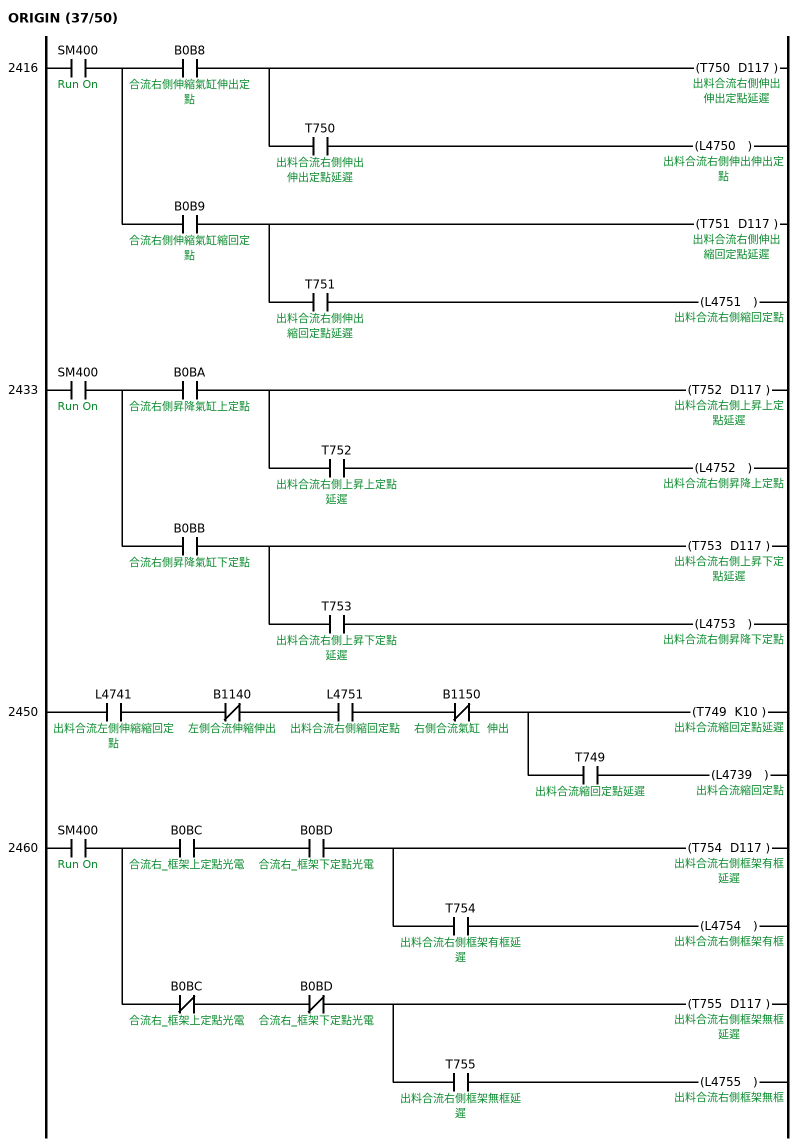
[picture p456: ladder of ORIGIN, rungs at steps 2416 to 2460]
2416  LD      SM400  ; Run On
      MPS
      AND     B0B8  ; 合流右側伸縮氣缸伸出定點
      OUT     T750 D117  ; 出料合流右側伸出 伸出定點延遲
      AND     T750  ; 出料合流右側伸出 伸出定點延遲
      OUT     L4750  ; 出料合流右側伸出伸出定點
      MPP
      AND     B0B9  ; 合流右側伸縮氣缸縮回定點
      OUT     T751 D117  ; 出料合流右側伸出 縮回定點延遲
      AND     T751  ; 出料合流右側伸出 縮回定點延遲
      OUT     L4751  ; 出料合流右側縮回定點
2433  LD      SM400  ; Run On
      MPS
      AND     B0BA  ; 合流右側昇降氣缸上定點
      OUT     T752 D117  ; 出料合流右側上昇上定點延遲
      AND     T752  ; 出料合流右側上昇上定點延遲
      OUT     L4752  ; 出料合流右側昇降上定點
      MPP
      AND     B0BB  ; 合流右側昇降氣缸下定點
      OUT     T753 D117  ; 出料合流右側上昇下定點延遲
      AND     T753  ; 出料合流右側上昇下定點延遲
      OUT     L4753  ; 出料合流右側昇降下定點
2450  LD      L4741  ; 出料合流左側伸縮縮回定點
      ANI     B1140  ; 左側合流伸縮伸出
      AND     L4751  ; 出料合流右側縮回定點
      ANI     B1150  ; 右側合流氣缸  伸出
      OUT     T749 K10  ; 出料合流縮回定點延遲
      AND     T749  ; 出料合流縮回定點延遲
      OUT     L4739  ; 出料合流縮回定點
2460  LD      SM400  ; Run On
      MPS
      AND     B0BC  ; 合流右_框架上定點光電
      AND     B0BD  ; 合流右_框架下定點光電
      OUT     T754 D117  ; 出料合流右側框架有框延遲
      AND     T754  ; 出料合流右側框架有框延遲
      OUT     L4754  ; 出料合流右側框架有框
      MPP
      ANI     B0BC  ; 合流右_框架上定點光電
      ANI     B0BD  ; 合流右_框架下定點光電
      OUT     T755 D117  ; 出料合流右側框架無框延遲
      AND     T755  ; 出料合流右側框架無框延遲
      OUT     L4755  ; 出料合流右側框架無框
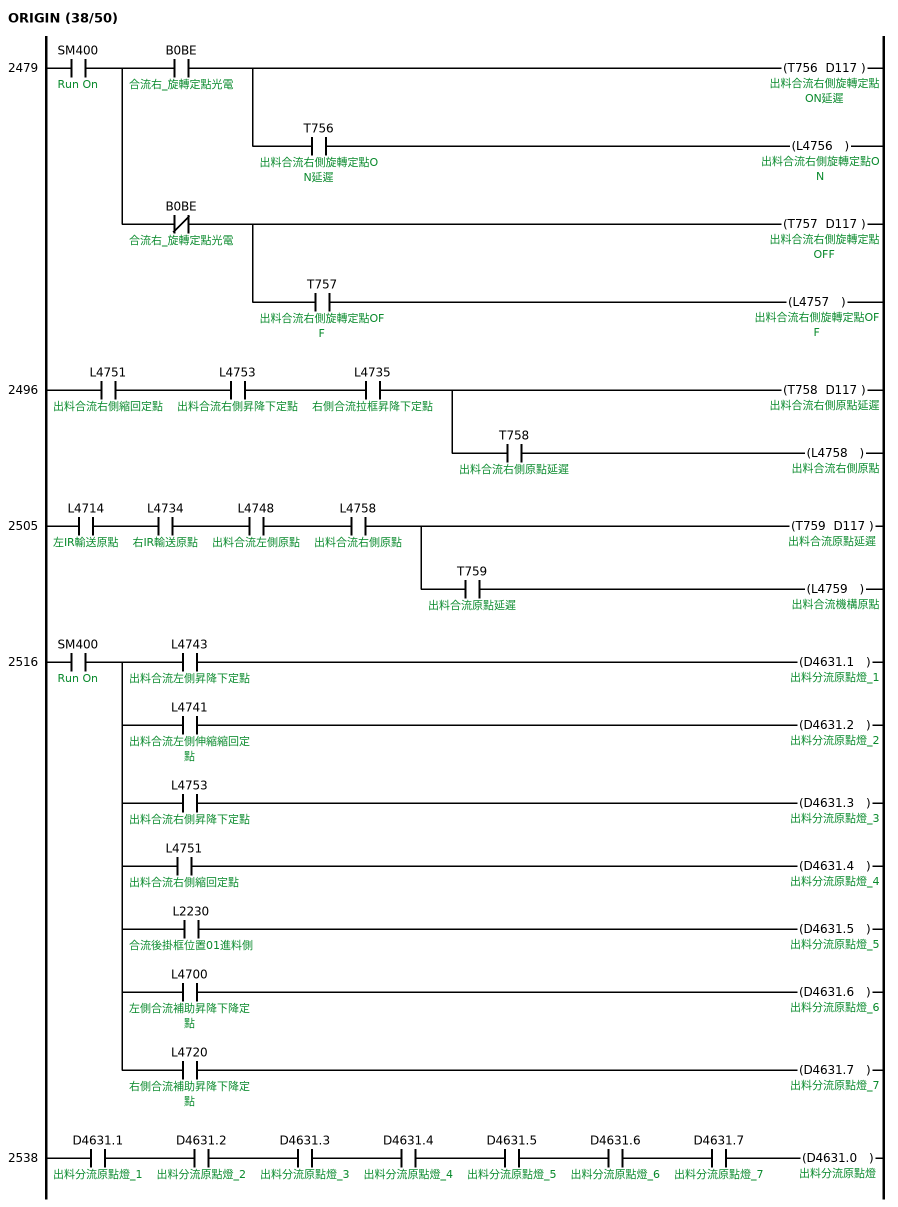
2479  LD      SM400  ; Run On
      MPS
      AND     B0BE  ; 合流右_旋轉定點光電
      OUT     T756 D117  ; 出料合流右側旋轉定點ON延遲
      AND     T756  ; 出料合流右側旋轉定點ON延遲
      OUT     L4756  ; 出料合流右側旋轉定點ON
      MPP
      ANI     B0BE  ; 合流右_旋轉定點光電
      OUT     T757 D117  ; 出料合流右側旋轉定點OFF
      AND     T757  ; 出料合流右側旋轉定點OFF
      OUT     L4757  ; 出料合流右側旋轉定點OFF
2496  LD      L4751  ; 出料合流右側縮回定點
      AND     L4753  ; 出料合流右側昇降下定點
      AND     L4735  ; 右側合流拉框昇降下定點
      OUT     T758 D117  ; 出料合流右側原點延遲
      AND     T758  ; 出料合流右側原點延遲
      OUT     L4758  ; 出料合流右側原點
2505  LD      L4714  ; 左IR輸送原點
      AND     L4734  ; 右IR輸送原點
      AND     L4748  ; 出料合流左側原點
      AND     L4758  ; 出料合流右側原點
      OUT     T759 D117  ; 出料合流原點延遲
      AND     T759  ; 出料合流原點延遲
      OUT     L4759  ; 出料合流機構原點
2516  LD      SM400  ; Run On
      MPS
      AND     L4743  ; 出料合流左側昇降下定點
      OUT     D4631.1  ; 出料分流原點燈_1
      MRD
      AND     L4741  ; 出料合流左側伸縮縮回定點
      OUT     D4631.2  ; 出料分流原點燈_2
      MRD
      AND     L4753  ; 出料合流右側昇降下定點
      OUT     D4631.3  ; 出料分流原點燈_3
      MRD
      AND     L4751  ; 出料合流右側縮回定點
      OUT     D4631.4  ; 出料分流原點燈_4
      MRD
      AND     L2230  ; 合流後掛框位置01進料側
      OUT     D4631.5  ; 出料分流原點燈_5
      MRD
      AND     L4700  ; 左側合流補助昇降下降定點
      OUT     D4631.6  ; 出料分流原點燈_6
      MPP
      AND     L4720  ; 右側合流補助昇降下降定點
      OUT     D4631.7  ; 出料分流原點燈_7
2538  LD      D4631.1  ; 出料分流原點燈_1
      AND     D4631.2  ; 出料分流原點燈_2
      AND     D4631.3  ; 出料分流原點燈_3
      AND     D4631.4  ; 出料分流原點燈_4
      AND     D4631.5  ; 出料分流原點燈_5
      AND     D4631.6  ; 出料分流原點燈_6
      AND     D4631.7  ; 出料分流原點燈_7
      OUT     D4631.0  ; 出料分流原點燈
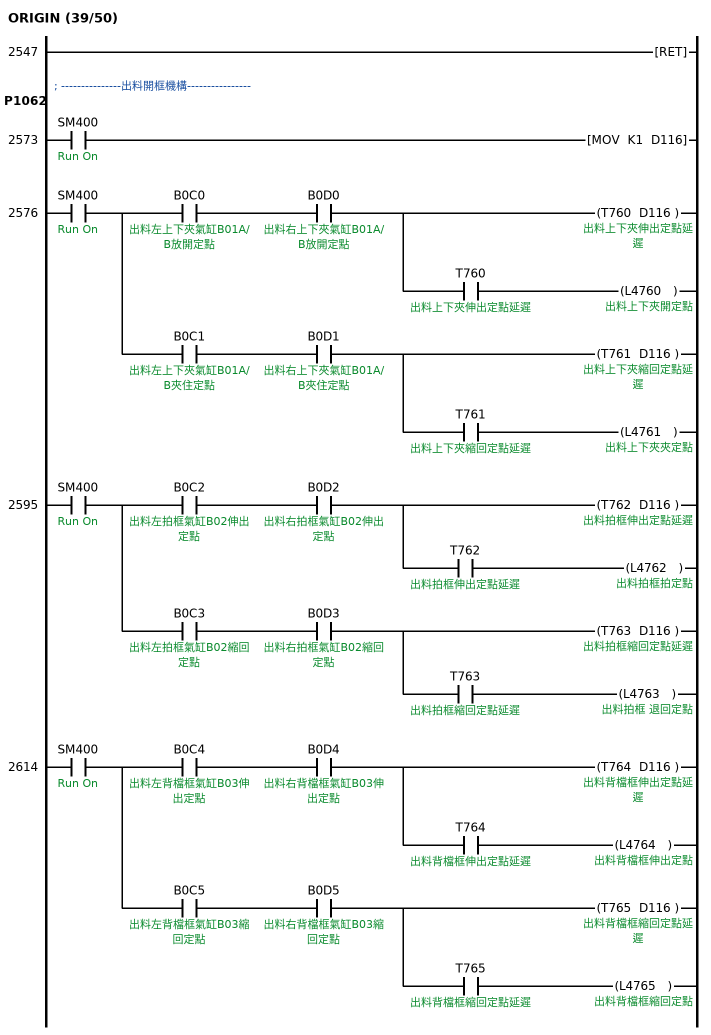
2547  RET
; ---------------出料開框機構----------------
      P1062
2573  LD      SM400  ; Run On
      MOV     K1 D116
2576  LD      SM400  ; Run On
      MPS
      AND     B0C0  ; 出料左上下夾氣缸B01A/B放開定點
      AND     B0D0  ; 出料右上下夾氣缸B01A/B放開定點
      OUT     T760 D116  ; 出料上下夾伸出定點延遲
      AND     T760  ; 出料上下夾伸出定點延遲
      OUT     L4760  ; 出料上下夾開定點
      MPP
      AND     B0C1  ; 出料左上下夾氣缸B01A/B夾住定點
      AND     B0D1  ; 出料右上下夾氣缸B01A/B夾住定點
      OUT     T761 D116  ; 出料上下夾縮回定點延遲
      AND     T761  ; 出料上下夾縮回定點延遲
      OUT     L4761  ; 出料上下夾夾定點
2595  LD      SM400  ; Run On
      MPS
      AND     B0C2  ; 出料左拍框氣缸B02伸出定點
      AND     B0D2  ; 出料右拍框氣缸B02伸出定點
      OUT     T762 D116  ; 出料拍框伸出定點延遲
      AND     T762  ; 出料拍框伸出定點延遲
      OUT     L4762  ; 出料拍框拍定點
      MPP
      AND     B0C3  ; 出料左拍框氣缸B02縮回定點
      AND     B0D3  ; 出料右拍框氣缸B02縮回定點
      OUT     T763 D116  ; 出料拍框縮回定點延遲
      AND     T763  ; 出料拍框縮回定點延遲
      OUT     L4763  ; 出料拍框 退回定點
2614  LD      SM400  ; Run On
      MPS
      AND     B0C4  ; 出料左背檔框氣缸B03伸出定點
      AND     B0D4  ; 出料右背檔框氣缸B03伸出定點
      OUT     T764 D116  ; 出料背檔框伸出定點延遲
      AND     T764  ; 出料背檔框伸出定點延遲
      OUT     L4764  ; 出料背檔框伸出定點
      MPP
      AND     B0C5  ; 出料左背檔框氣缸B03縮回定點
      AND     B0D5  ; 出料右背檔框氣缸B03縮回定點
      OUT     T765 D116  ; 出料背檔框縮回定點延遲
      AND     T765  ; 出料背檔框縮回定點延遲
      OUT     L4765  ; 出料背檔框縮回定點
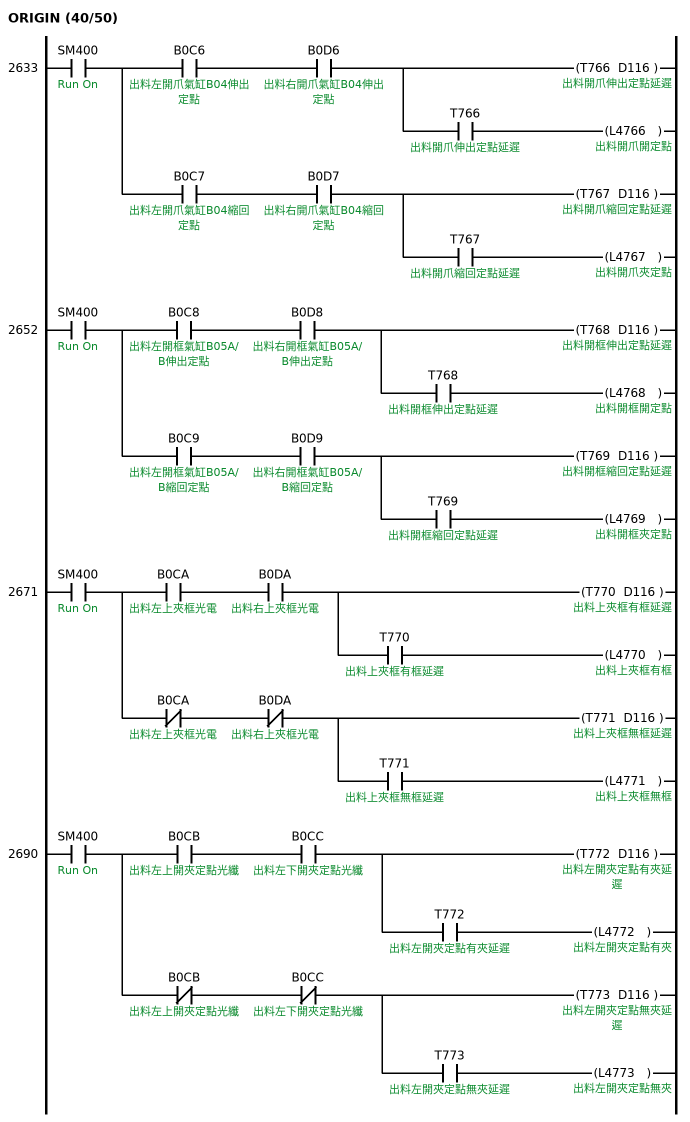
2633  LD      SM400  ; Run On
      MPS
      AND     B0C6  ; 出料左開爪氣缸B04伸出定點
      AND     B0D6  ; 出料右開爪氣缸B04伸出定點
      OUT     T766 D116  ; 出料開爪伸出定點延遲
      AND     T766  ; 出料開爪伸出定點延遲
      OUT     L4766  ; 出料開爪開定點
      MPP
      AND     B0C7  ; 出料左開爪氣缸B04縮回定點
      AND     B0D7  ; 出料右開爪氣缸B04縮回定點
      OUT     T767 D116  ; 出料開爪縮回定點延遲
      AND     T767  ; 出料開爪縮回定點延遲
      OUT     L4767  ; 出料開爪夾定點
2652  LD      SM400  ; Run On
      MPS
      AND     B0C8  ; 出料左開框氣缸B05A/B伸出定點
      AND     B0D8  ; 出料右開框氣缸B05A/B伸出定點
      OUT     T768 D116  ; 出料開框伸出定點延遲
      AND     T768  ; 出料開框伸出定點延遲
      OUT     L4768  ; 出料開框開定點
      MPP
      AND     B0C9  ; 出料左開框氣缸B05A/B縮回定點
      AND     B0D9  ; 出料右開框氣缸B05A/B縮回定點
      OUT     T769 D116  ; 出料開框縮回定點延遲
      AND     T769  ; 出料開框縮回定點延遲
      OUT     L4769  ; 出料開框夾定點
2671  LD      SM400  ; Run On
      MPS
      AND     B0CA  ; 出料左上夾框光電
      AND     B0DA  ; 出料右上夾框光電
      OUT     T770 D116  ; 出料上夾框有框延遲
      AND     T770  ; 出料上夾框有框延遲
      OUT     L4770  ; 出料上夾框有框
      MPP
      ANI     B0CA  ; 出料左上夾框光電
      ANI     B0DA  ; 出料右上夾框光電
      OUT     T771 D116  ; 出料上夾框無框延遲
      AND     T771  ; 出料上夾框無框延遲
      OUT     L4771  ; 出料上夾框無框
2690  LD      SM400  ; Run On
      MPS
      AND     B0CB  ; 出料左上開夾定點光纖
      AND     B0CC  ; 出料左下開夾定點光纖
      OUT     T772 D116  ; 出料左開夾定點有夾延遲
      AND     T772  ; 出料左開夾定點有夾延遲
      OUT     L4772  ; 出料左開夾定點有夾
      MPP
      ANI     B0CB  ; 出料左上開夾定點光纖
      ANI     B0CC  ; 出料左下開夾定點光纖
      OUT     T773 D116  ; 出料左開夾定點無夾延遲
      AND     T773  ; 出料左開夾定點無夾延遲
      OUT     L4773  ; 出料左開夾定點無夾
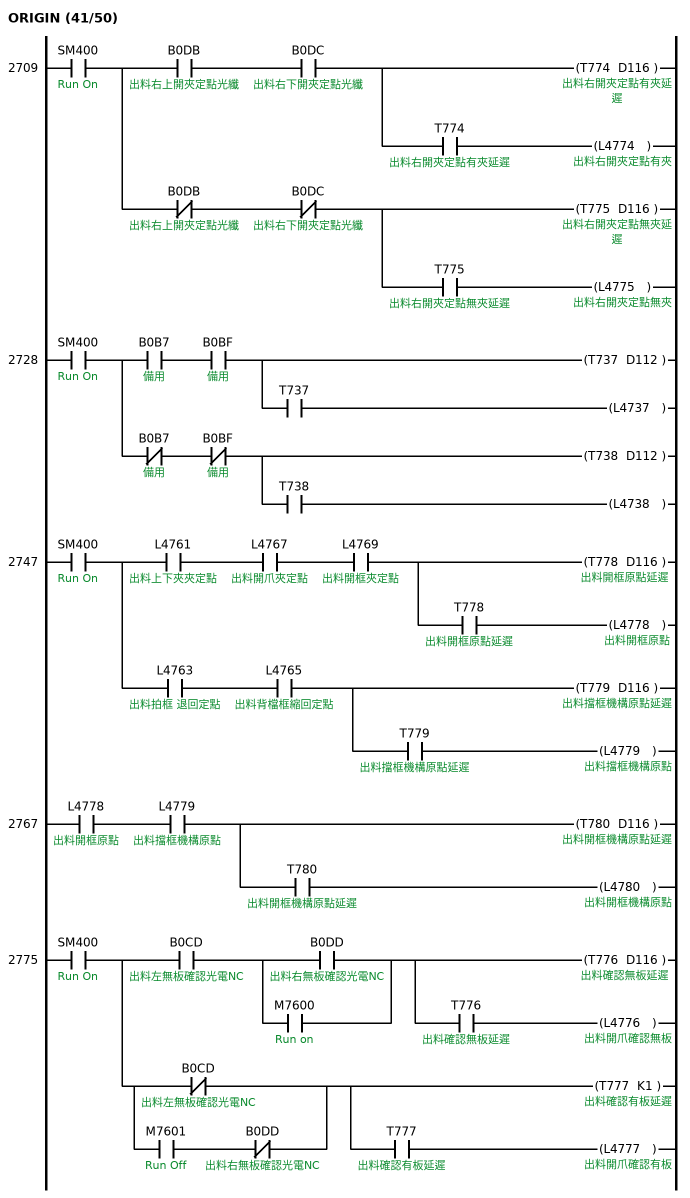
2709  LD      SM400  ; Run On
      MPS
      AND     B0DB  ; 出料右上開夾定點光纖
      AND     B0DC  ; 出料右下開夾定點光纖
      OUT     T774 D116  ; 出料右開夾定點有夾延遲
      AND     T774  ; 出料右開夾定點有夾延遲
      OUT     L4774  ; 出料右開夾定點有夾
      MPP
      ANI     B0DB  ; 出料右上開夾定點光纖
      ANI     B0DC  ; 出料右下開夾定點光纖
      OUT     T775 D116  ; 出料右開夾定點無夾延遲
      AND     T775  ; 出料右開夾定點無夾延遲
      OUT     L4775  ; 出料右開夾定點無夾
2728  LD      SM400  ; Run On
      MPS
      AND     B0B7  ; 備用
      AND     B0BF  ; 備用
      OUT     T737 D112
      AND     T737
      OUT     L4737
      MPP
      ANI     B0B7  ; 備用
      ANI     B0BF  ; 備用
      OUT     T738 D112
      AND     T738
      OUT     L4738
2747  LD      SM400  ; Run On
      MPS
      AND     L4761  ; 出料上下夾夾定點
      AND     L4767  ; 出料開爪夾定點
      AND     L4769  ; 出料開框夾定點
      OUT     T778 D116  ; 出料開框原點延遲
      AND     T778  ; 出料開框原點延遲
      OUT     L4778  ; 出料開框原點
      MPP
      AND     L4763  ; 出料拍框 退回定點
      AND     L4765  ; 出料背檔框縮回定點
      OUT     T779 D116  ; 出料擋框機構原點延遲
      AND     T779  ; 出料擋框機構原點延遲
      OUT     L4779  ; 出料擋框機構原點
2767  LD      L4778  ; 出料開框原點
      AND     L4779  ; 出料擋框機構原點
      OUT     T780 D116  ; 出料開框機構原點延遲
      AND     T780  ; 出料開框機構原點延遲
      OUT     L4780  ; 出料開框機構原點
2775  LD      SM400  ; Run On
      MPS
      AND     B0CD  ; 出料左無板確認光電NC
      LD      B0DD  ; 出料右無板確認光電NC
      OR      M7600  ; Run on
      ANB
      OUT     T776 D116  ; 出料確認無板延遲
      AND     T776  ; 出料確認無板延遲
      OUT     L4776  ; 出料開爪確認無板
      MPP
      LDI     B0CD  ; 出料左無板確認光電NC
      LD      M7601  ; Run Off
      ANI     B0DD  ; 出料右無板確認光電NC
      ORB
      ANB
      OUT     T777 K1  ; 出料確認有板延遲
      AND     T777  ; 出料確認有板延遲
      OUT     L4777  ; 出料開爪確認有板
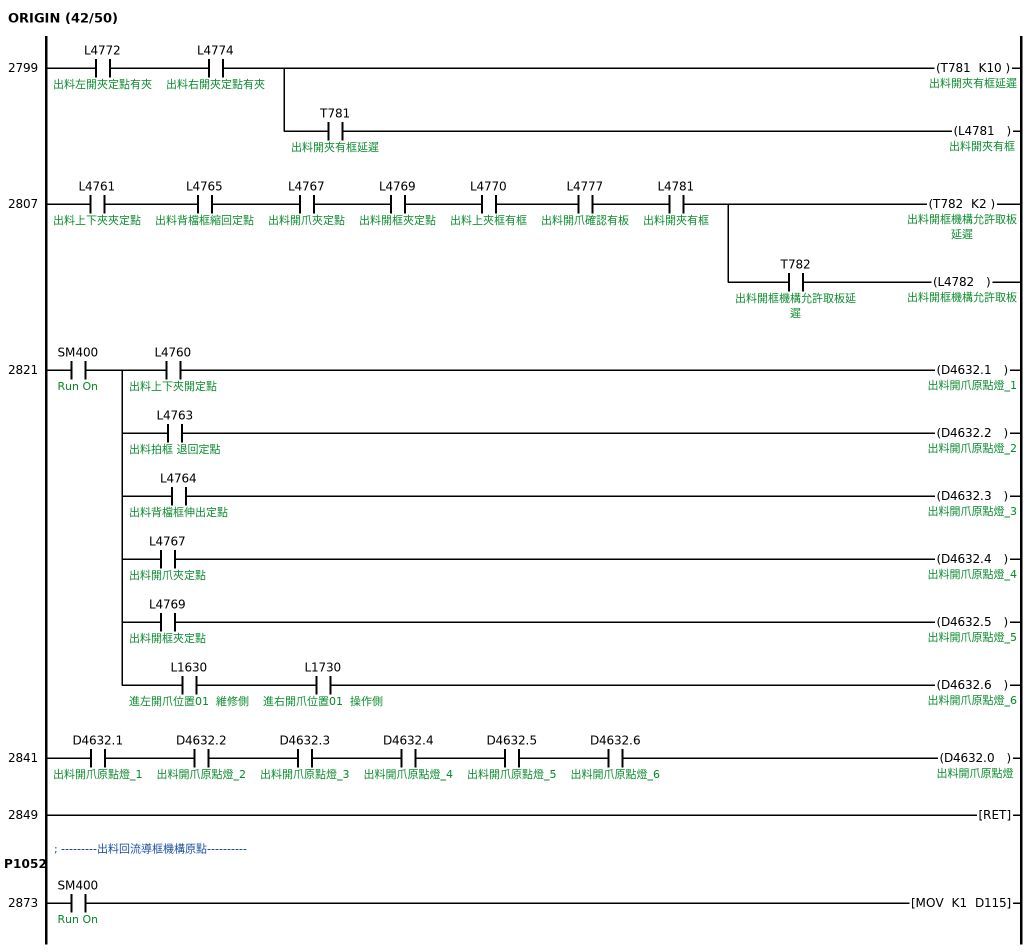
2799  LD      L4772  ; 出料左開夾定點有夾
      AND     L4774  ; 出料右開夾定點有夾
      OUT     T781 K10  ; 出料開夾有框延遲
      AND     T781  ; 出料開夾有框延遲
      OUT     L4781  ; 出料開夾有框
2807  LD      L4761  ; 出料上下夾夾定點
      AND     L4765  ; 出料背檔框縮回定點
      AND     L4767  ; 出料開爪夾定點
      AND     L4769  ; 出料開框夾定點
      AND     L4770  ; 出料上夾框有框
      AND     L4777  ; 出料開爪確認有板
      AND     L4781  ; 出料開夾有框
      OUT     T782 K2  ; 出料開框機構允許取板延遲
      AND     T782  ; 出料開框機構允許取板延遲
      OUT     L4782  ; 出料開框機構允許取板
2821  LD      SM400  ; Run On
      MPS
      AND     L4760  ; 出料上下夾開定點
      OUT     D4632.1  ; 出料開爪原點燈_1
      MRD
      AND     L4763  ; 出料拍框 退回定點
      OUT     D4632.2  ; 出料開爪原點燈_2
      MRD
      AND     L4764  ; 出料背檔框伸出定點
      OUT     D4632.3  ; 出料開爪原點燈_3
      MRD
      AND     L4767  ; 出料開爪夾定點
      OUT     D4632.4  ; 出料開爪原點燈_4
      MRD
      AND     L4769  ; 出料開框夾定點
      OUT     D4632.5  ; 出料開爪原點燈_5
      MPP
      AND     L1630  ; 進左開爪位置01  維修側
      AND     L1730  ; 進右開爪位置01  操作側
      OUT     D4632.6  ; 出料開爪原點燈_6
2841  LD      D4632.1  ; 出料開爪原點燈_1
      AND     D4632.2  ; 出料開爪原點燈_2
      AND     D4632.3  ; 出料開爪原點燈_3
      AND     D4632.4  ; 出料開爪原點燈_4
      AND     D4632.5  ; 出料開爪原點燈_5
      AND     D4632.6  ; 出料開爪原點燈_6
      OUT     D4632.0  ; 出料開爪原點燈
2849  RET
; ---------出料回流導框機構原點----------
      P1052
2873  LD      SM400  ; Run On
      MOV     K1 D115
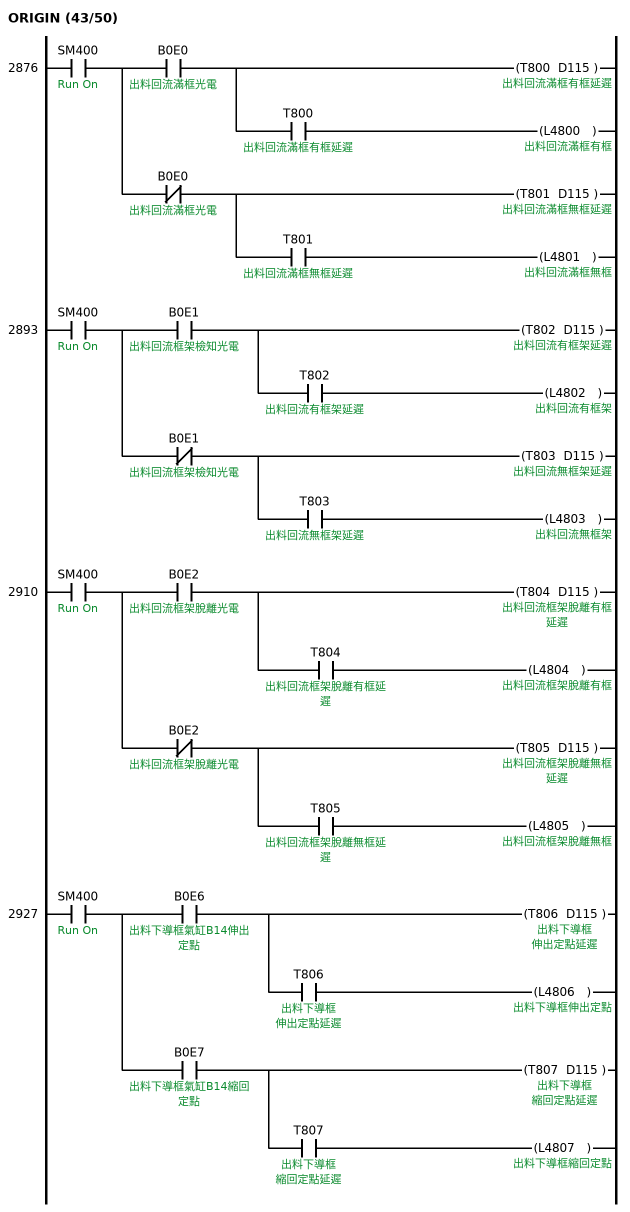
2876  LD      SM400  ; Run On
      MPS
      AND     B0E0  ; 出料回流滿框光電
      OUT     T800 D115  ; 出料回流滿框有框延遲
      AND     T800  ; 出料回流滿框有框延遲
      OUT     L4800  ; 出料回流滿框有框
      MPP
      ANI     B0E0  ; 出料回流滿框光電
      OUT     T801 D115  ; 出料回流滿框無框延遲
      AND     T801  ; 出料回流滿框無框延遲
      OUT     L4801  ; 出料回流滿框無框
2893  LD      SM400  ; Run On
      MPS
      AND     B0E1  ; 出料回流框架檢知光電
      OUT     T802 D115  ; 出料回流有框架延遲
      AND     T802  ; 出料回流有框架延遲
      OUT     L4802  ; 出料回流有框架
      MPP
      ANI     B0E1  ; 出料回流框架檢知光電
      OUT     T803 D115  ; 出料回流無框架延遲
      AND     T803  ; 出料回流無框架延遲
      OUT     L4803  ; 出料回流無框架
2910  LD      SM400  ; Run On
      MPS
      AND     B0E2  ; 出料回流框架脫離光電
      OUT     T804 D115  ; 出料回流框架脫離有框延遲
      AND     T804  ; 出料回流框架脫離有框延遲
      OUT     L4804  ; 出料回流框架脫離有框
      MPP
      ANI     B0E2  ; 出料回流框架脫離光電
      OUT     T805 D115  ; 出料回流框架脫離無框延遲
      AND     T805  ; 出料回流框架脫離無框延遲
      OUT     L4805  ; 出料回流框架脫離無框
2927  LD      SM400  ; Run On
      MPS
      AND     B0E6  ; 出料下導框氣缸B14伸出定點
      OUT     T806 D115  ; 出料下導框    伸出定點延遲
      AND     T806  ; 出料下導框    伸出定點延遲
      OUT     L4806  ; 出料下導框伸出定點
      MPP
      AND     B0E7  ; 出料下導框氣缸B14縮回定點
      OUT     T807 D115  ; 出料下導框    縮回定點延遲
      AND     T807  ; 出料下導框    縮回定點延遲
      OUT     L4807  ; 出料下導框縮回定點
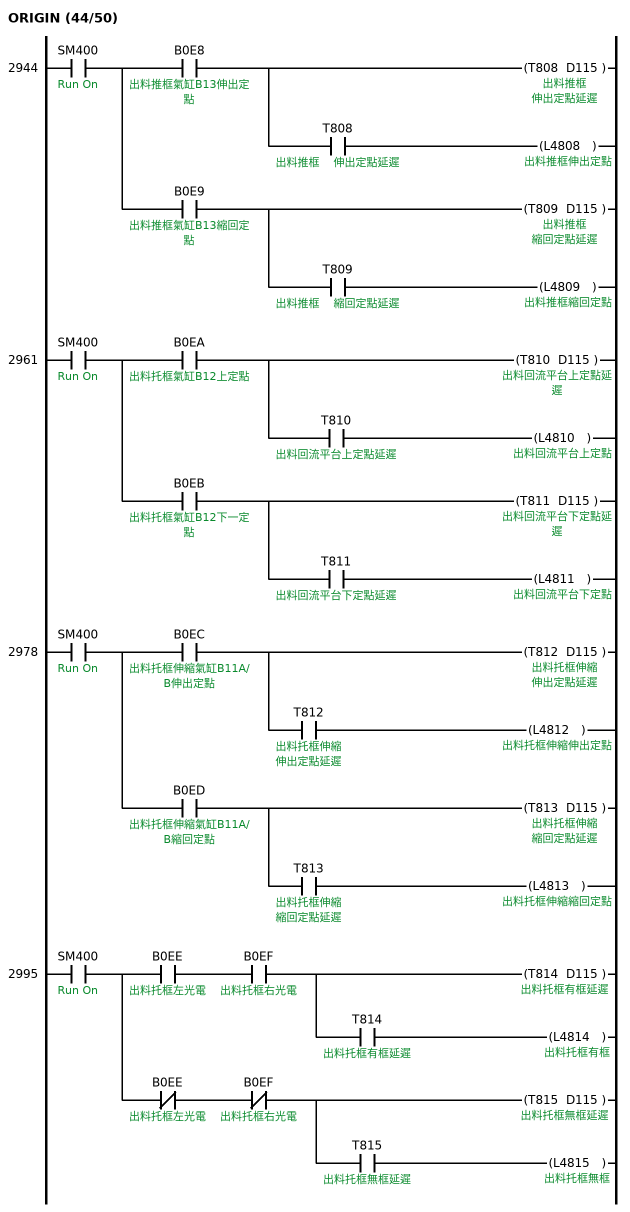
2944  LD      SM400  ; Run On
      MPS
      AND     B0E8  ; 出料推框氣缸B13伸出定點
      OUT     T808 D115  ; 出料推框    伸出定點延遲
      AND     T808  ; 出料推框    伸出定點延遲
      OUT     L4808  ; 出料推框伸出定點
      MPP
      AND     B0E9  ; 出料推框氣缸B13縮回定點
      OUT     T809 D115  ; 出料推框    縮回定點延遲
      AND     T809  ; 出料推框    縮回定點延遲
      OUT     L4809  ; 出料推框縮回定點
2961  LD      SM400  ; Run On
      MPS
      AND     B0EA  ; 出料托框氣缸B12上定點
      OUT     T810 D115  ; 出料回流平台上定點延遲
      AND     T810  ; 出料回流平台上定點延遲
      OUT     L4810  ; 出料回流平台上定點
      MPP
      AND     B0EB  ; 出料托框氣缸B12下一定點
      OUT     T811 D115  ; 出料回流平台下定點延遲
      AND     T811  ; 出料回流平台下定點延遲
      OUT     L4811  ; 出料回流平台下定點
2978  LD      SM400  ; Run On
      MPS
      AND     B0EC  ; 出料托框伸縮氣缸B11A/B伸出定點
      OUT     T812 D115  ; 出料托框伸縮    伸出定點延遲
      AND     T812  ; 出料托框伸縮    伸出定點延遲
      OUT     L4812  ; 出料托框伸縮伸出定點
      MPP
      AND     B0ED  ; 出料托框伸縮氣缸B11A/B縮回定點
      OUT     T813 D115  ; 出料托框伸縮    縮回定點延遲
      AND     T813  ; 出料托框伸縮    縮回定點延遲
      OUT     L4813  ; 出料托框伸縮縮回定點
2995  LD      SM400  ; Run On
      MPS
      AND     B0EE  ; 出料托框左光電
      AND     B0EF  ; 出料托框右光電
      OUT     T814 D115  ; 出料托框有框延遲
      AND     T814  ; 出料托框有框延遲
      OUT     L4814  ; 出料托框有框
      MPP
      ANI     B0EE  ; 出料托框左光電
      ANI     B0EF  ; 出料托框右光電
      OUT     T815 D115  ; 出料托框無框延遲
      AND     T815  ; 出料托框無框延遲
      OUT     L4815  ; 出料托框無框
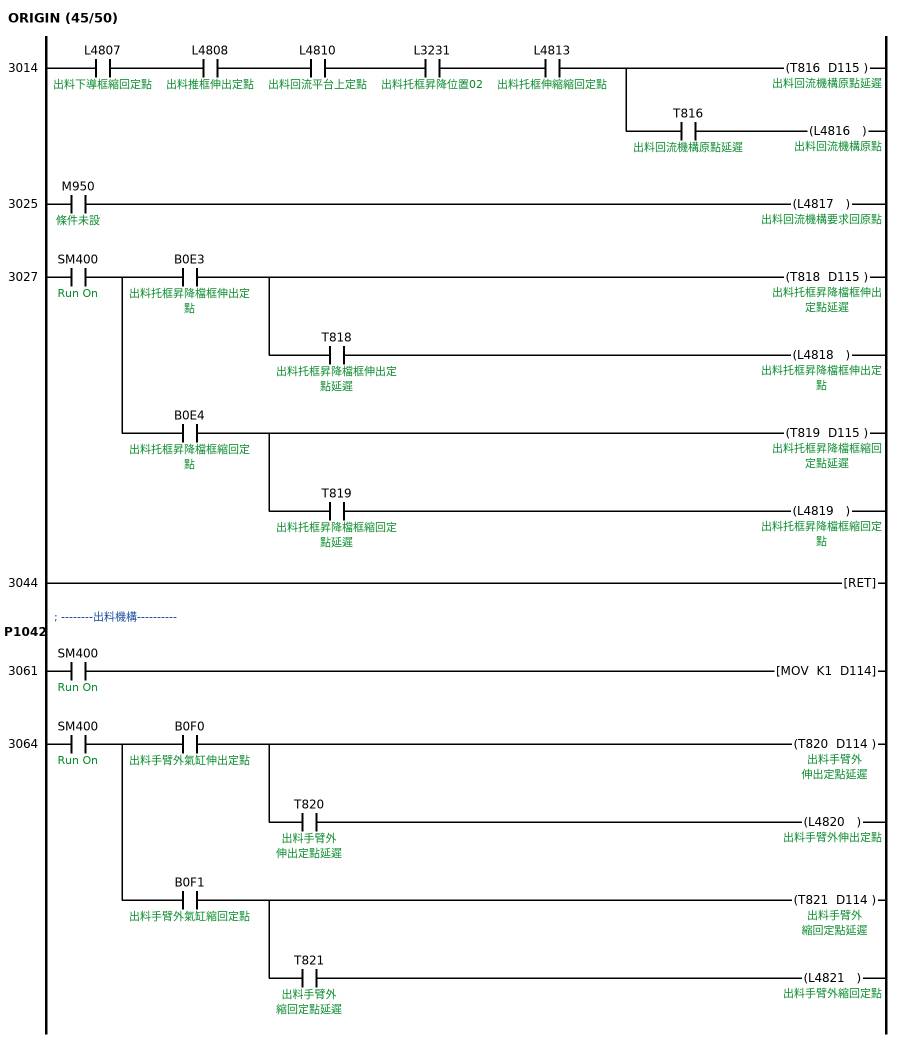
3014  LD      L4807  ; 出料下導框縮回定點
      AND     L4808  ; 出料推框伸出定點
      AND     L4810  ; 出料回流平台上定點
      AND     L3231  ; 出料托框昇降位置02
      AND     L4813  ; 出料托框伸縮縮回定點
      OUT     T816 D115  ; 出料回流機構原點延遲
      AND     T816  ; 出料回流機構原點延遲
      OUT     L4816  ; 出料回流機構原點
3025  LD      M950  ; 條件未設
      OUT     L4817  ; 出料回流機構要求回原點
3027  LD      SM400  ; Run On
      MPS
      AND     B0E3  ; 出料托框昇降檔框伸出定點
      OUT     T818 D115  ; 出料托框昇降檔框伸出定點延遲
      AND     T818  ; 出料托框昇降檔框伸出定點延遲
      OUT     L4818  ; 出料托框昇降檔框伸出定點
      MPP
      AND     B0E4  ; 出料托框昇降檔框縮回定點
      OUT     T819 D115  ; 出料托框昇降檔框縮回定點延遲
      AND     T819  ; 出料托框昇降檔框縮回定點延遲
      OUT     L4819  ; 出料托框昇降檔框縮回定點
3044  RET
; --------出料機構----------
      P1042
3061  LD      SM400  ; Run On
      MOV     K1 D114
3064  LD      SM400  ; Run On
      MPS
      AND     B0F0  ; 出料手臂外氣缸伸出定點
      OUT     T820 D114  ; 出料手臂外    伸出定點延遲
      AND     T820  ; 出料手臂外    伸出定點延遲
      OUT     L4820  ; 出料手臂外伸出定點
      MPP
      AND     B0F1  ; 出料手臂外氣缸縮回定點
      OUT     T821 D114  ; 出料手臂外    縮回定點延遲
      AND     T821  ; 出料手臂外    縮回定點延遲
      OUT     L4821  ; 出料手臂外縮回定點
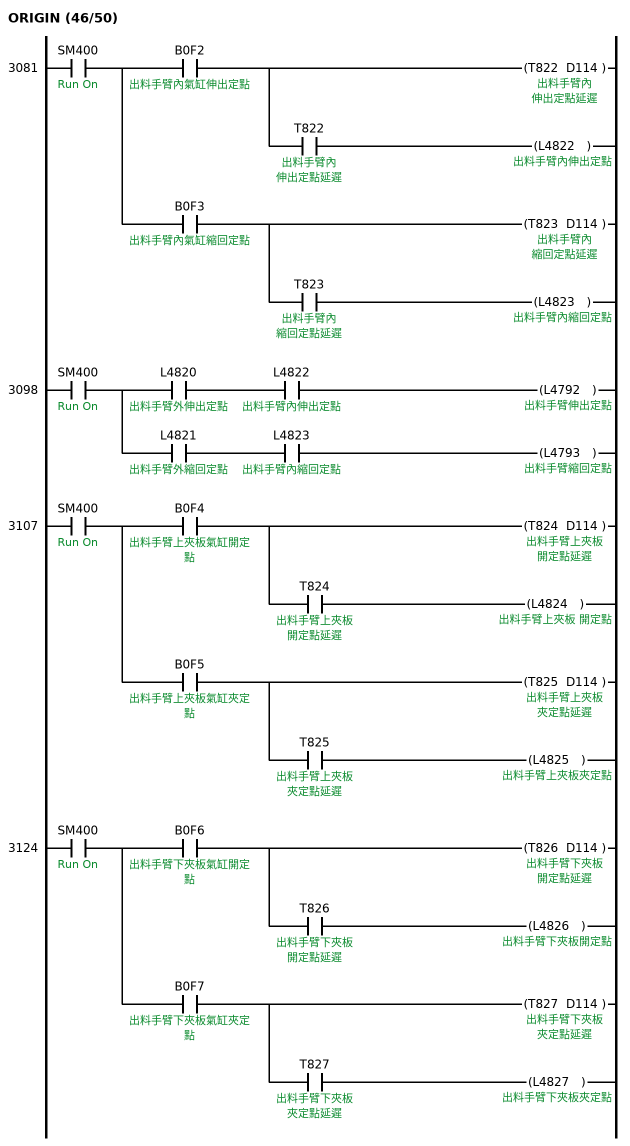
3081  LD      SM400  ; Run On
      MPS
      AND     B0F2  ; 出料手臂內氣缸伸出定點
      OUT     T822 D114  ; 出料手臂內    伸出定點延遲
      AND     T822  ; 出料手臂內    伸出定點延遲
      OUT     L4822  ; 出料手臂內伸出定點
      MPP
      AND     B0F3  ; 出料手臂內氣缸縮回定點
      OUT     T823 D114  ; 出料手臂內    縮回定點延遲
      AND     T823  ; 出料手臂內    縮回定點延遲
      OUT     L4823  ; 出料手臂內縮回定點
3098  LD      SM400  ; Run On
      MPS
      AND     L4820  ; 出料手臂外伸出定點
      AND     L4822  ; 出料手臂內伸出定點
      OUT     L4792  ; 出料手臂伸出定點
      MPP
      AND     L4821  ; 出料手臂外縮回定點
      AND     L4823  ; 出料手臂內縮回定點
      OUT     L4793  ; 出料手臂縮回定點
3107  LD      SM400  ; Run On
      MPS
      AND     B0F4  ; 出料手臂上夾板氣缸開定點
      OUT     T824 D114  ; 出料手臂上夾板    開定點延遲
      AND     T824  ; 出料手臂上夾板    開定點延遲
      OUT     L4824  ; 出料手臂上夾板 開定點
      MPP
      AND     B0F5  ; 出料手臂上夾板氣缸夾定點
      OUT     T825 D114  ; 出料手臂上夾板    夾定點延遲
      AND     T825  ; 出料手臂上夾板    夾定點延遲
      OUT     L4825  ; 出料手臂上夾板夾定點
3124  LD      SM400  ; Run On
      MPS
      AND     B0F6  ; 出料手臂下夾板氣缸開定點
      OUT     T826 D114  ; 出料手臂下夾板    開定點延遲
      AND     T826  ; 出料手臂下夾板    開定點延遲
      OUT     L4826  ; 出料手臂下夾板開定點
      MPP
      AND     B0F7  ; 出料手臂下夾板氣缸夾定點
      OUT     T827 D114  ; 出料手臂下夾板    夾定點延遲
      AND     T827  ; 出料手臂下夾板    夾定點延遲
      OUT     L4827  ; 出料手臂下夾板夾定點
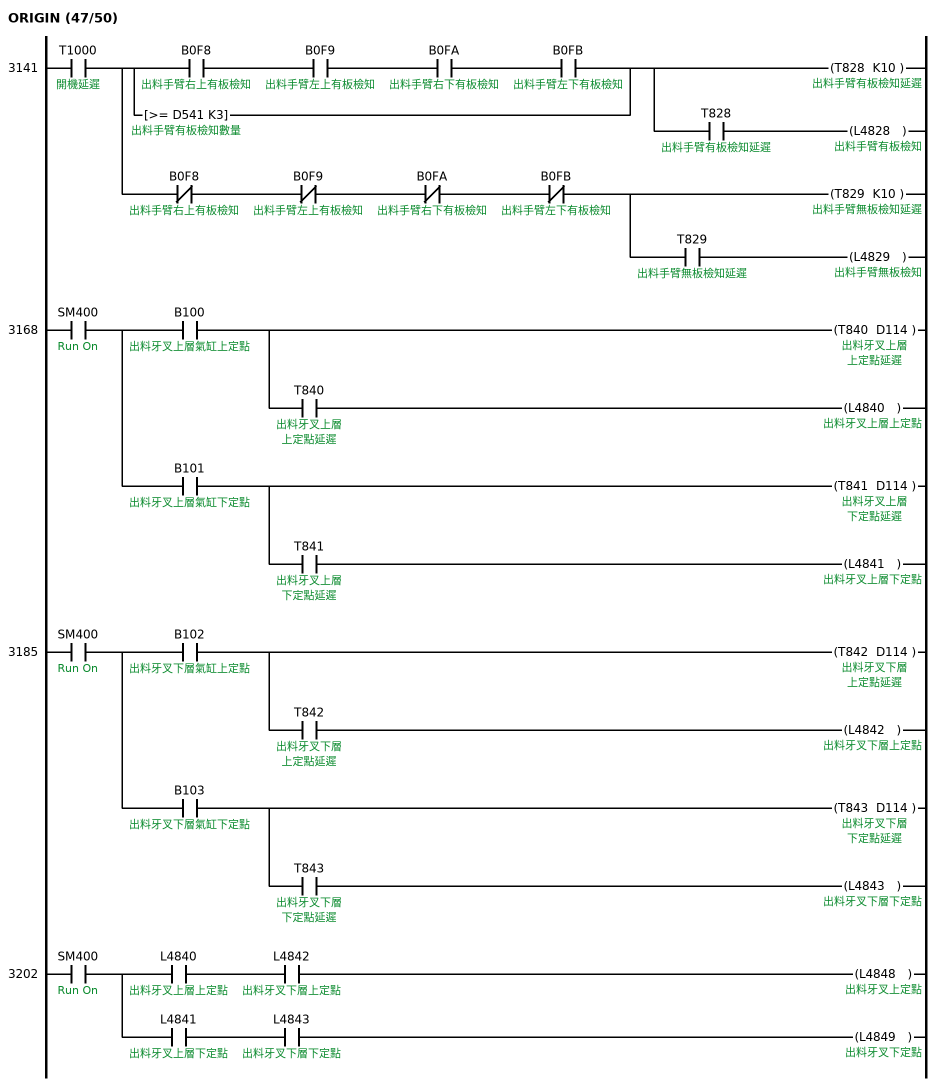
3141  LD      T1000  ; 開機延遲
      MPS
      LD      B0F8  ; 出料手臂右上有板檢知
      AND     B0F9  ; 出料手臂左上有板檢知
      AND     B0FA  ; 出料手臂右下有板檢知
      AND     B0FB  ; 出料手臂左下有板檢知
      OR>=    D541 K3  ; 出料手臂有板檢知數量
      ANB
      OUT     T828 K10  ; 出料手臂有板檢知延遲
      AND     T828  ; 出料手臂有板檢知延遲
      OUT     L4828  ; 出料手臂有板檢知
      MPP
      ANI     B0F8  ; 出料手臂右上有板檢知
      ANI     B0F9  ; 出料手臂左上有板檢知
      ANI     B0FA  ; 出料手臂右下有板檢知
      ANI     B0FB  ; 出料手臂左下有板檢知
      OUT     T829 K10  ; 出料手臂無板檢知延遲
      AND     T829  ; 出料手臂無板檢知延遲
      OUT     L4829  ; 出料手臂無板檢知
3168  LD      SM400  ; Run On
      MPS
      AND     B100  ; 出料牙叉上層氣缸上定點
      OUT     T840 D114  ; 出料牙叉上層    上定點延遲
      AND     T840  ; 出料牙叉上層    上定點延遲
      OUT     L4840  ; 出料牙叉上層上定點
      MPP
      AND     B101  ; 出料牙叉上層氣缸下定點
      OUT     T841 D114  ; 出料牙叉上層    下定點延遲
      AND     T841  ; 出料牙叉上層    下定點延遲
      OUT     L4841  ; 出料牙叉上層下定點
3185  LD      SM400  ; Run On
      MPS
      AND     B102  ; 出料牙叉下層氣缸上定點
      OUT     T842 D114  ; 出料牙叉下層    上定點延遲
      AND     T842  ; 出料牙叉下層    上定點延遲
      OUT     L4842  ; 出料牙叉下層上定點
      MPP
      AND     B103  ; 出料牙叉下層氣缸下定點
      OUT     T843 D114  ; 出料牙叉下層    下定點延遲
      AND     T843  ; 出料牙叉下層    下定點延遲
      OUT     L4843  ; 出料牙叉下層下定點
3202  LD      SM400  ; Run On
      MPS
      AND     L4840  ; 出料牙叉上層上定點
      AND     L4842  ; 出料牙叉下層上定點
      OUT     L4848  ; 出料牙叉上定點
      MPP
      AND     L4841  ; 出料牙叉上層下定點
      AND     L4843  ; 出料牙叉下層下定點
      OUT     L4849  ; 出料牙叉下定點
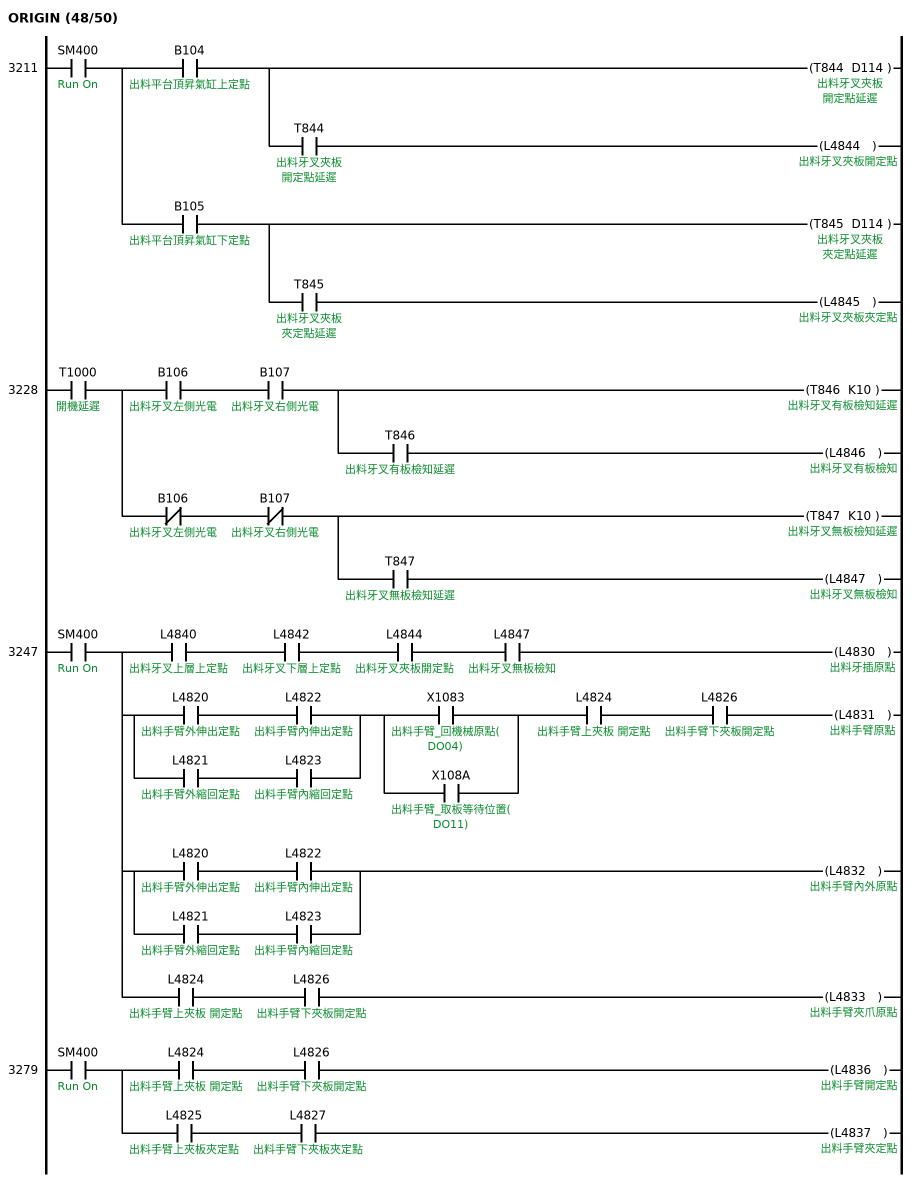
3211  LD      SM400  ; Run On
      MPS
      AND     B104  ; 出料平台頂昇氣缸上定點
      OUT     T844 D114  ; 出料牙叉夾板    開定點延遲
      AND     T844  ; 出料牙叉夾板    開定點延遲
      OUT     L4844  ; 出料牙叉夾板開定點
      MPP
      AND     B105  ; 出料平台頂昇氣缸下定點
      OUT     T845 D114  ; 出料牙叉夾板    夾定點延遲
      AND     T845  ; 出料牙叉夾板    夾定點延遲
      OUT     L4845  ; 出料牙叉夾板夾定點
3228  LD      T1000  ; 開機延遲
      MPS
      AND     B106  ; 出料牙叉左側光電
      AND     B107  ; 出料牙叉右側光電
      OUT     T846 K10  ; 出料牙叉有板檢知延遲
      AND     T846  ; 出料牙叉有板檢知延遲
      OUT     L4846  ; 出料牙叉有板檢知
      MPP
      ANI     B106  ; 出料牙叉左側光電
      ANI     B107  ; 出料牙叉右側光電
      OUT     T847 K10  ; 出料牙叉無板檢知延遲
      AND     T847  ; 出料牙叉無板檢知延遲
      OUT     L4847  ; 出料牙叉無板檢知
3247  LD      SM400  ; Run On
      MPS
      AND     L4840  ; 出料牙叉上層上定點
      AND     L4842  ; 出料牙叉下層上定點
      AND     L4844  ; 出料牙叉夾板開定點
      AND     L4847  ; 出料牙叉無板檢知
      OUT     L4830  ; 出料牙插原點
      MRD
      LD      L4820  ; 出料手臂外伸出定點
      AND     L4822  ; 出料手臂內伸出定點
      LD      L4821  ; 出料手臂外縮回定點
      AND     L4823  ; 出料手臂內縮回定點
      ORB
      ANB
      LD      X1083  ; 出料手臂_回機械原點(DO04)
      OR      X108A  ; 出料手臂_取板等待位置(DO11)
      ANB
      AND     L4824  ; 出料手臂上夾板 開定點
      AND     L4826  ; 出料手臂下夾板開定點
      OUT     L4831  ; 出料手臂原點
      MRD
      LD      L4820  ; 出料手臂外伸出定點
      AND     L4822  ; 出料手臂內伸出定點
      LD      L4821  ; 出料手臂外縮回定點
      AND     L4823  ; 出料手臂內縮回定點
      ORB
      ANB
      OUT     L4832  ; 出料手臂內外原點
      MPP
      AND     L4824  ; 出料手臂上夾板 開定點
      AND     L4826  ; 出料手臂下夾板開定點
      OUT     L4833  ; 出料手臂夾爪原點
3279  LD      SM400  ; Run On
      MPS
      AND     L4824  ; 出料手臂上夾板 開定點
      AND     L4826  ; 出料手臂下夾板開定點
      OUT     L4836  ; 出料手臂開定點
      MPP
      AND     L4825  ; 出料手臂上夾板夾定點
      AND     L4827  ; 出料手臂下夾板夾定點
      OUT     L4837  ; 出料手臂夾定點
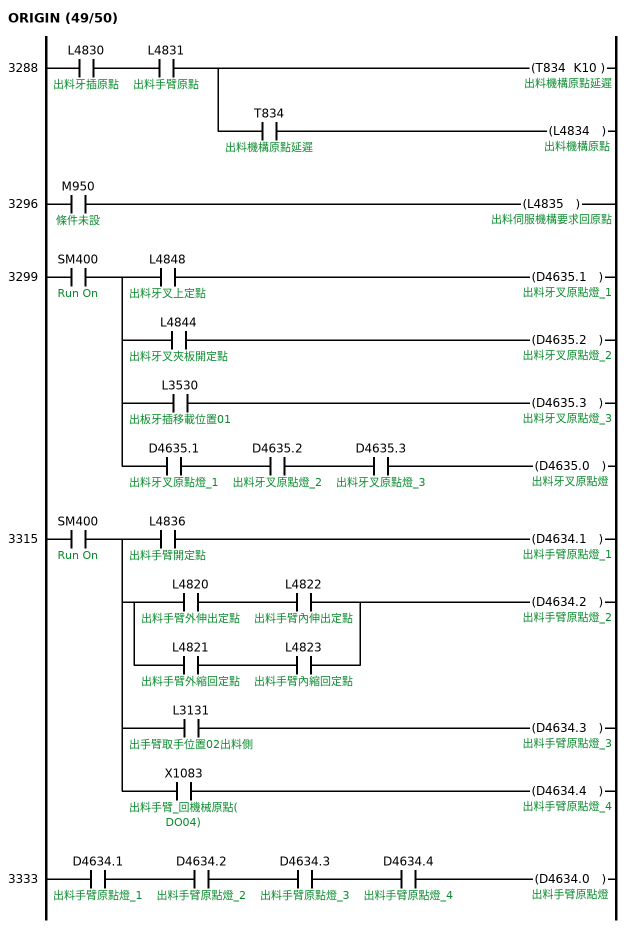
3288  LD      L4830  ; 出料牙插原點
      AND     L4831  ; 出料手臂原點
      OUT     T834 K10  ; 出料機構原點延遲
      AND     T834  ; 出料機構原點延遲
      OUT     L4834  ; 出料機構原點
3296  LD      M950  ; 條件未設
      OUT     L4835  ; 出料伺服機構要求回原點
3299  LD      SM400  ; Run On
      MPS
      AND     L4848  ; 出料牙叉上定點
      OUT     D4635.1  ; 出料牙叉原點燈_1
      MRD
      AND     L4844  ; 出料牙叉夾板開定點
      OUT     D4635.2  ; 出料牙叉原點燈_2
      MRD
      AND     L3530  ; 出板牙插移載位置01
      OUT     D4635.3  ; 出料牙叉原點燈_3
      MPP
      AND     D4635.1  ; 出料牙叉原點燈_1
      AND     D4635.2  ; 出料牙叉原點燈_2
      AND     D4635.3  ; 出料牙叉原點燈_3
      OUT     D4635.0  ; 出料牙叉原點燈
3315  LD      SM400  ; Run On
      MPS
      AND     L4836  ; 出料手臂開定點
      OUT     D4634.1  ; 出料手臂原點燈_1
      MRD
      LD      L4820  ; 出料手臂外伸出定點
      AND     L4822  ; 出料手臂內伸出定點
      LD      L4821  ; 出料手臂外縮回定點
      AND     L4823  ; 出料手臂內縮回定點
      ORB
      ANB
      OUT     D4634.2  ; 出料手臂原點燈_2
      MRD
      AND     L3131  ; 出手臂取手位置02出料側
      OUT     D4634.3  ; 出料手臂原點燈_3
      MPP
      AND     X1083  ; 出料手臂_回機械原點(DO04)
      OUT     D4634.4  ; 出料手臂原點燈_4
3333  LD      D4634.1  ; 出料手臂原點燈_1
      AND     D4634.2  ; 出料手臂原點燈_2
      AND     D4634.3  ; 出料手臂原點燈_3
      AND     D4634.4  ; 出料手臂原點燈_4
      OUT     D4634.0  ; 出料手臂原點燈
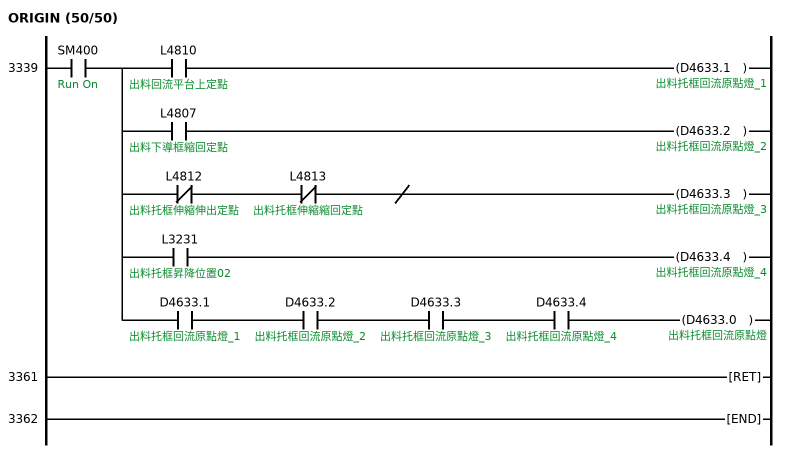
3339  LD      SM400  ; Run On
      MPS
      AND     L4810  ; 出料回流平台上定點
      OUT     D4633.1  ; 出料托框回流原點燈_1
      MRD
      AND     L4807  ; 出料下導框縮回定點
      OUT     D4633.2  ; 出料托框回流原點燈_2
      MRD
      ANI     L4812  ; 出料托框伸縮伸出定點
      ANI     L4813  ; 出料托框伸縮縮回定點
      INV
      OUT     D4633.3  ; 出料托框回流原點燈_3
      MRD
      AND     L3231  ; 出料托框昇降位置02
      OUT     D4633.4  ; 出料托框回流原點燈_4
      MPP
      AND     D4633.1  ; 出料托框回流原點燈_1
      AND     D4633.2  ; 出料托框回流原點燈_2
      AND     D4633.3  ; 出料托框回流原點燈_3
      AND     D4633.4  ; 出料托框回流原點燈_4
      OUT     D4633.0  ; 出料托框回流原點燈
3361  RET
3362  END
END_PROGRAM

PROGRAM SECS
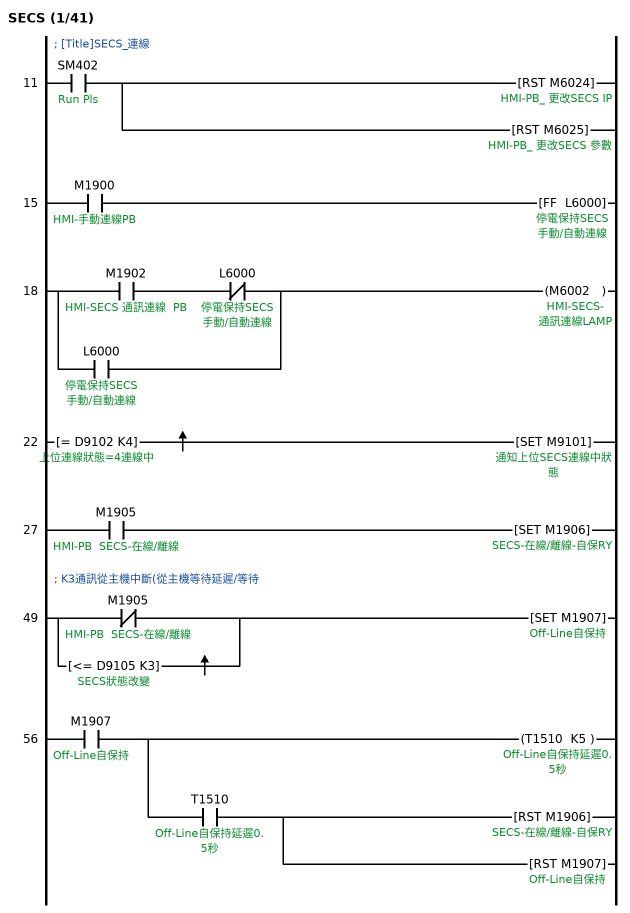
; [Title]SECS_連線
11    LD      SM402  ; Run Pls
      RST     M6024  ; HMI-PB_ 更改SECS IP
      RST     M6025  ; HMI-PB_ 更改SECS 參數
15    LD      M1900  ; HMI-手動連線PB
      FF      L6000  ; 停電保持SECS    手動/自動連線
18    LD      M1902  ; HMI-SECS 通訊連線  PB
      ANI     L6000  ; 停電保持SECS    手動/自動連線
      OR      L6000  ; 停電保持SECS    手動/自動連線
      OUT     M6002  ; HMI-SECS- 通訊連線LAMP
22    LD=     D9102 K4  ; 上位連線狀態=4連線中
      MEP
      SET     M9101  ; 通知上位SECS連線中狀態
27    LD      M1905  ; HMI-PB  SECS-在線/離線
      SET     M1906  ; SECS-在線/離線-自保RY
; K3通訊從主機中斷(從主機等待延遲/等待
49    LDI     M1905  ; HMI-PB  SECS-在線/離線
      LD<=    D9105 K3  ; SECS狀態改變
      MEP
      ORB
      SET     M1907  ; Off-Line自保持
56    LD      M1907  ; Off-Line自保持
      OUT     T1510 K5  ; Off-Line自保持延遲0.5秒
      AND     T1510  ; Off-Line自保持延遲0.5秒
      RST     M1906  ; SECS-在線/離線-自保RY
      RST     M1907  ; Off-Line自保持
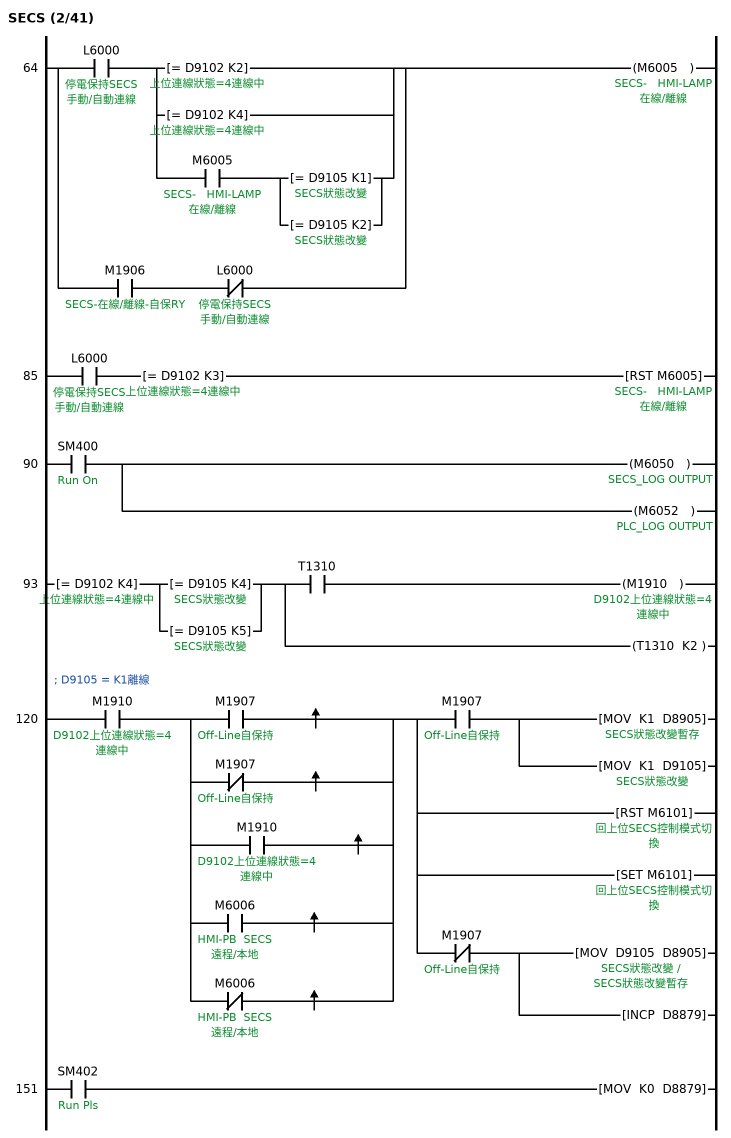
64    LD      L6000  ; 停電保持SECS    手動/自動連線
      LD=     D9102 K2  ; 上位連線狀態=4連線中
      OR=     D9102 K4  ; 上位連線狀態=4連線中
      LD      M6005  ; SECS-   HMI-LAMP 在線/離線
      LD=     D9105 K1  ; SECS狀態改變
      OR=     D9105 K2  ; SECS狀態改變
      ANB
      ORB
      ANB
      LD      M1906  ; SECS-在線/離線-自保RY
      ANI     L6000  ; 停電保持SECS    手動/自動連線
      ORB
      OUT     M6005  ; SECS-   HMI-LAMP 在線/離線
85    LD      L6000  ; 停電保持SECS    手動/自動連線
      AND=    D9102 K3  ; 上位連線狀態=4連線中
      RST     M6005  ; SECS-   HMI-LAMP 在線/離線
90    LD      SM400  ; Run On
      OUT     M6050  ; SECS_LOG OUTPUT
      OUT     M6052  ; PLC_LOG OUTPUT
93    LD=     D9102 K4  ; 上位連線狀態=4連線中
      LD=     D9105 K4  ; SECS狀態改變
      OR=     D9105 K5  ; SECS狀態改變
      ANB
      MPS
      AND     T1310
      OUT     M1910  ; D9102上位連線狀態=4連線中
      MPP
      OUT     T1310 K2
; D9105 = K1離線
120   LD      M1910  ; D9102上位連線狀態=4連線中
      LD      M1907  ; Off-Line自保持
      MEP
      LDI     M1907  ; Off-Line自保持
      MEP
      ORB
      LD      M1910  ; D9102上位連線狀態=4連線中
      MEP
      ORB
      LD      M6006  ; HMI-PB  SECS  遠程/本地
      MEP
      ORB
      LDI     M6006  ; HMI-PB  SECS  遠程/本地
      MEP
      ORB
      ANB
      MPS
      AND     M1907  ; Off-Line自保持
      MOV     K1 D8905  ; SECS狀態改變暫存
      MOV     K1 D9105
      MPP
      RST     M6101  ; 回上位SECS控制模式切換
      SET     M6101  ; 回上位SECS控制模式切換
      ANI     M1907  ; Off-Line自保持
      MOV     D9105 D8905
      INCP    D8879
151   LD      SM402  ; Run Pls
      MOV     K0 D8879
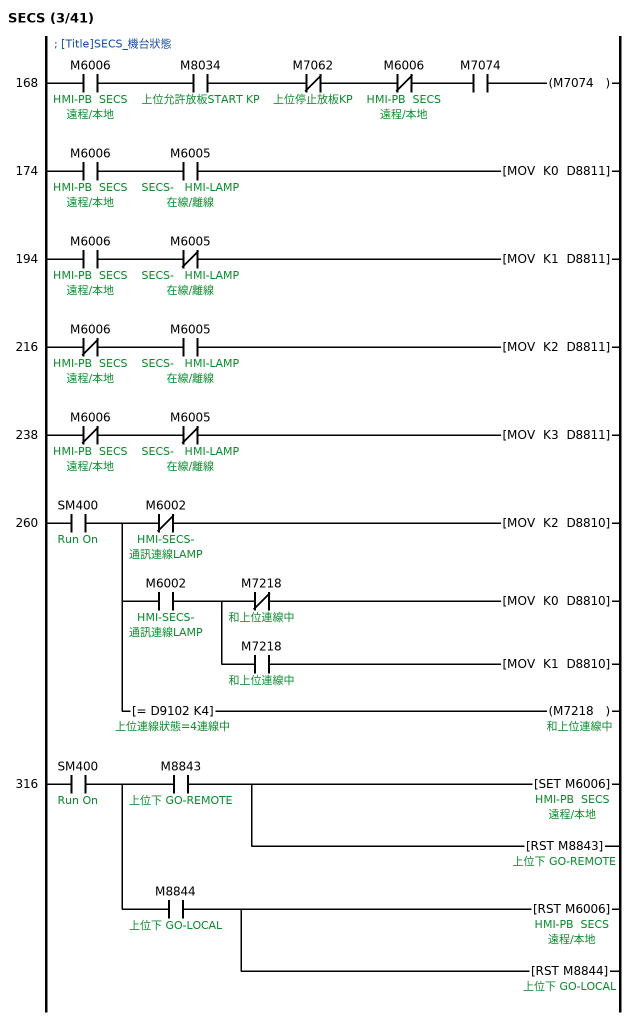
; [Title]SECS_機台狀態
168   LD      M6006  ; HMI-PB  SECS  遠程/本地
      AND     M8034  ; 上位允許放板START KP
      ANI     M7062  ; 上位停止放板KP
      ANI     M6006  ; HMI-PB  SECS  遠程/本地
      AND     M7074
      OUT     M7074
174   LD      M6006  ; HMI-PB  SECS  遠程/本地
      AND     M6005  ; SECS-   HMI-LAMP 在線/離線
      MOV     K0 D8811
        [note] D8811=K0(遠程控制+SEC在線中)
194   LD      M6006  ; HMI-PB  SECS  遠程/本地
      ANI     M6005  ; SECS-   HMI-LAMP 在線/離線
      MOV     K1 D8811
        [note] D8811= k1(遠程控制中+SEC離線中)
216   LDI     M6006  ; HMI-PB  SECS  遠程/本地
      AND     M6005  ; SECS-   HMI-LAMP 在線/離線
      MOV     K2 D8811
        [note] D881=k2(遠程控制離線+SEC在線中)
238   LDI     M6006  ; HMI-PB  SECS  遠程/本地
      ANI     M6005  ; SECS-   HMI-LAMP 在線/離線
      MOV     K3 D8811
        [note] D881=k3(遠程控制離線+SEC離線中)
260   LD      SM400  ; Run On
      MPS
      ANI     M6002  ; HMI-SECS- 通訊連線LAMP
      MOV     K2 D8810
        [note] K2= SEC通訊未連線
      MRD
      AND     M6002  ; HMI-SECS- 通訊連線LAMP
      MPS
      ANI     M7218  ; 和上位連線中
      MOV     K0 D8810
        [note] K0=SEC連線---上位未連線
      MPP
      AND     M7218  ; 和上位連線中
      MOV     K1 D8810
        [note] K1=SEC和上位連線中
      MPP
      AND=    D9102 K4  ; 上位連線狀態=4連線中
      OUT     M7218  ; 和上位連線中
316   LD      SM400  ; Run On
      MPS
      AND     M8843  ; 上位下 GO-REMOTE
      SET     M6006  ; HMI-PB  SECS  遠程/本地
      RST     M8843  ; 上位下 GO-REMOTE
      MPP
      AND     M8844  ; 上位下 GO-LOCAL
      RST     M6006  ; HMI-PB  SECS  遠程/本地
      RST     M8844  ; 上位下 GO-LOCAL
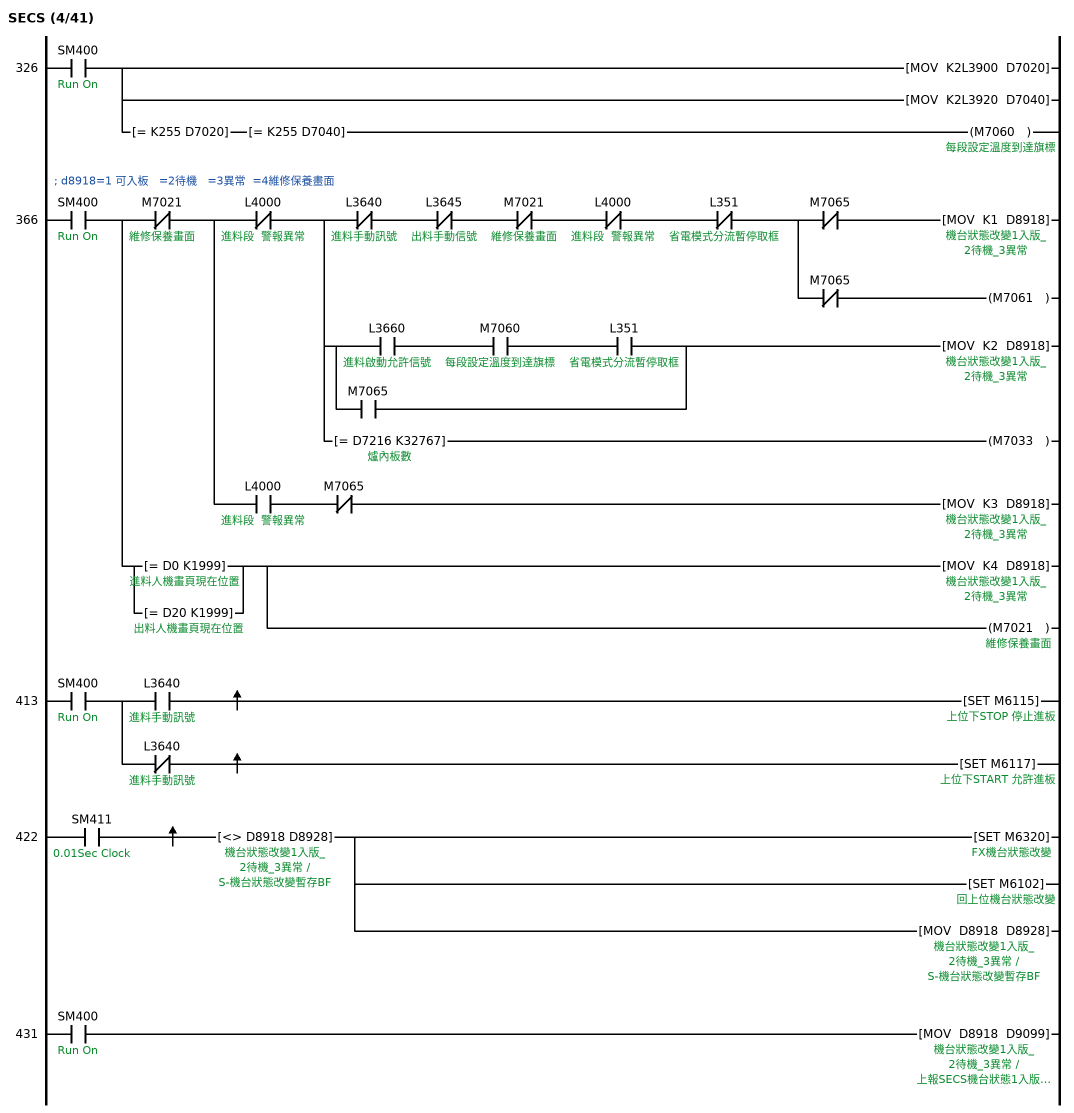
326   LD      SM400  ; Run On
      MOV     K2L3900 D7020  ; 溫度到達H01
      MOV     K2L3920 D7040  ; 溫度到達IRA01
      AND=    K255 D7020
      AND=    K255 D7040
      OUT     M7060  ; 每段設定溫度到達旗標
; d8918=1 可入板   =2待機   =3異常  =4維修保養畫面
366   LD      SM400  ; Run On
      MPS
      ANI     M7021  ; 維修保養畫面
      MPS
      ANI     L4000  ; 進料段  警報異常
      MPS
      ANI     L3640  ; 進料手動訊號
      ANI     L3645  ; 出料手動信號
      ANI     M7021  ; 維修保養畫面
      ANI     L4000  ; 進料段  警報異常
      ANI     L351  ; 省電模式分流暫停取框
      MPS
      ANI     M7065
      MOV     K1 D8918  ; 機台狀態改變1入版_2待機_3異常
      MPP
      ANI     M7065
      OUT     M7061
      MRD
      LD      L3660  ; 進料啟動允許信號
      AND     M7060  ; 每段設定溫度到達旗標
      AND     L351  ; 省電模式分流暫停取框
      OR      M7065
      ANB
      MOV     K2 D8918
      MPP
      AND=    D7216 K32767  ; 爐內板數
      OUT     M7033
      MPP
      AND     L4000  ; 進料段  警報異常
      ANI     M7065
      MOV     K3 D8918
      MPP
      LD=     D0 K1999  ; 進料人機畫頁現在位置
      OR=     D20 K1999  ; 出料人機畫頁現在位置
      ANB
      MOV     K4 D8918
      OUT     M7021  ; 維修保養畫面
413   LD      SM400  ; Run On
      MPS
      AND     L3640  ; 進料手動訊號
      MEP
      SET     M6115  ; 上位下STOP 停止進板
      MPP
      ANI     L3640  ; 進料手動訊號
      MEP
      SET     M6117  ; 上位下START 允許進板
422   LD      SM411  ; 0.01Sec Clock
      MEP
      AND<>   D8918 D8928  ; 機台狀態改變1入版_2待機_3異常 / S-機台狀態改變暫存BF
      SET     M6320  ; FX機台狀態改變
      SET     M6102  ; 回上位機台狀態改變
      MOV     D8918 D8928
431   LD      SM400  ; Run On
      MOV     D8918 D9099  ; 上報SECS機台狀態1入版_2待機_3異
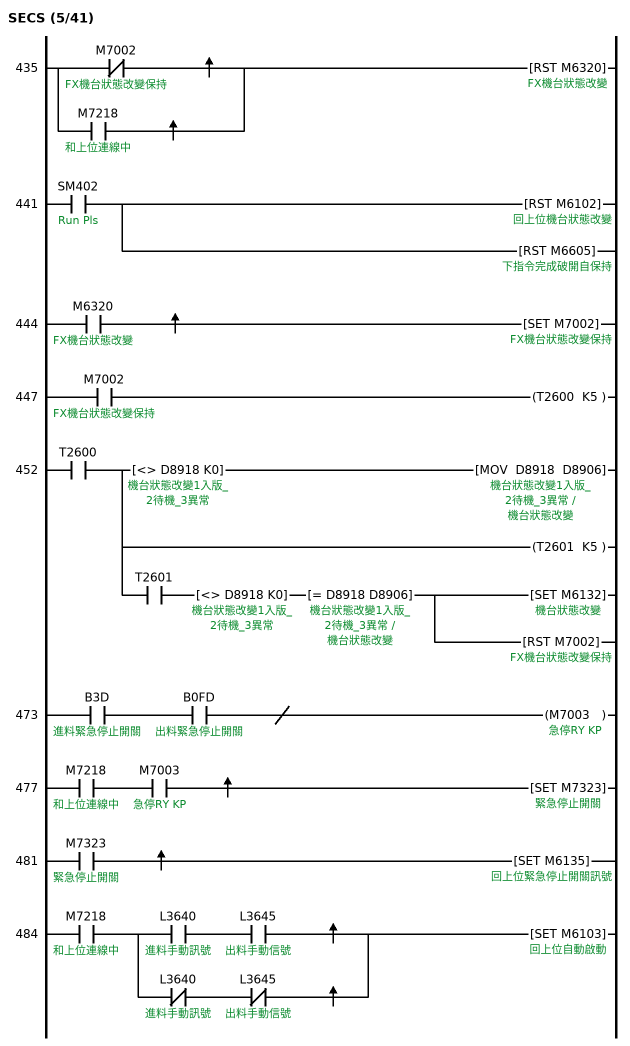
435   LDI     M7002  ; FX機台狀態改變保持
      MEP
      LD      M7218  ; 和上位連線中
      MEP
      ORB
      RST     M6320  ; FX機台狀態改變
441   LD      SM402  ; Run Pls
      RST     M6102  ; 回上位機台狀態改變
      RST     M6605  ; 下指令完成破開自保持
444   LD      M6320  ; FX機台狀態改變
      MEP
      SET     M7002  ; FX機台狀態改變保持
447   LD      M7002  ; FX機台狀態改變保持
      OUT     T2600 K5
452   LD      T2600
      MPS
      AND<>   D8918 K0  ; 機台狀態改變1入版_2待機_3異常
      MOV     D8918 D8906  ; 機台狀態改變
      MPP
      OUT     T2601 K5
      AND     T2601
      AND<>   D8918 K0  ; 機台狀態改變1入版_2待機_3異常
      AND=    D8918 D8906  ; 機台狀態改變1入版_2待機_3異常 / 機台狀態改變
      SET     M6132  ; 機台狀態改變
      RST     M7002  ; FX機台狀態改變保持
473   LD      B3D  ; 進料緊急停止開關
      AND     B0FD  ; 出料緊急停止開關
      INV
      OUT     M7003  ; 急停RY KP
477   LD      M7218  ; 和上位連線中
      AND     M7003  ; 急停RY KP
      MEP
      SET     M7323  ; 緊急停止開關
481   LD      M7323  ; 緊急停止開關
      MEP
      SET     M6135  ; 回上位緊急停止開關訊號
484   LD      M7218  ; 和上位連線中
      LD      L3640  ; 進料手動訊號
      AND     L3645  ; 出料手動信號
      MEP
      LDI     L3640  ; 進料手動訊號
      ANI     L3645  ; 出料手動信號
      MEP
      ORB
      ANB
      SET     M6103  ; 回上位自動啟動
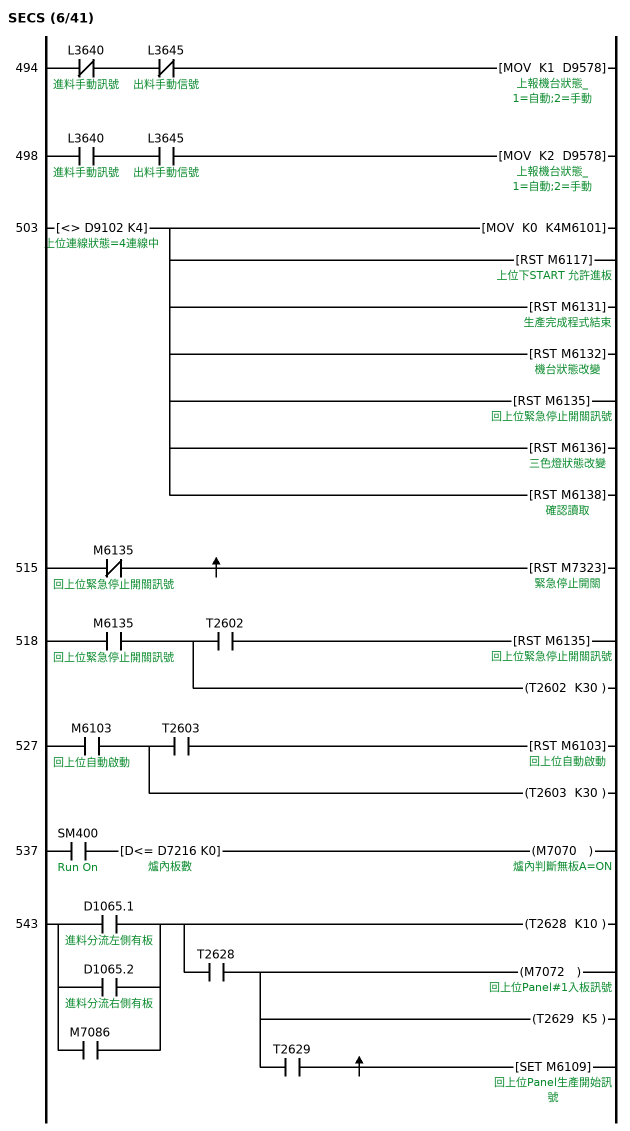
494   LDI     L3640  ; 進料手動訊號
      ANI     L3645  ; 出料手動信號
      MOV     K1 D9578  ; 上報機台狀態_1=自動;2=手動
498   LD      L3640  ; 進料手動訊號
      AND     L3645  ; 出料手動信號
      MOV     K2 D9578
503   LD<>    D9102 K4  ; 上位連線狀態=4連線中
      MOV     K0 K4M6101
      RST     M6117  ; 上位下START 允許進板
      RST     M6131  ; 生產完成程式結束
      RST     M6132  ; 機台狀態改變
      RST     M6135  ; 回上位緊急停止開關訊號
      RST     M6136  ; 三色燈狀態改變
      RST     M6138  ; 確認讀取
515   LDI     M6135  ; 回上位緊急停止開關訊號
      MEP
      RST     M7323  ; 緊急停止開關
518   LD      M6135  ; 回上位緊急停止開關訊號
      MPS
      AND     T2602
      RST     M6135  ; 回上位緊急停止開關訊號
      MPP
      OUT     T2602 K30
527   LD      M6103  ; 回上位自動啟動
      MPS
      AND     T2603
      RST     M6103  ; 回上位自動啟動
      MPP
      OUT     T2603 K30
537   LD      SM400  ; Run On
      ANDD<=  D7216 K0  ; 爐內板數
      OUT     M7070  ; 爐內判斷無板A=ON
543   LD      D1065.1  ; 進料分流左側有板
      OR      D1065.2  ; 進料分流右側有板
      OR      M7086
      OUT     T2628 K10
      AND     T2628
      OUT     M7072  ; 回上位Panel#1入板訊號
      OUT     T2629 K5
      AND     T2629
      MEP
      SET     M6109  ; 回上位Panel生產開始訊號
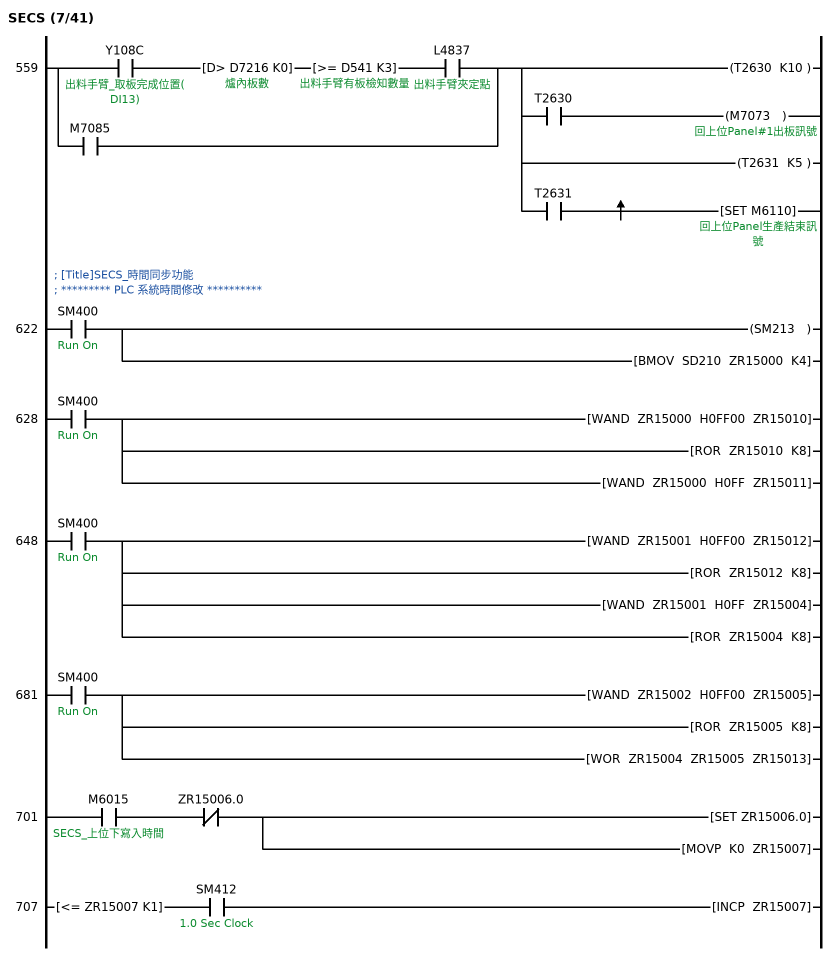
559   LD      Y108C  ; 出料手臂_取板完成位置(DI13)
      ANDD>   D7216 K0  ; 爐內板數
      AND>=   D541 K3  ; 出料手臂有板檢知數量
      AND     L4837  ; 出料手臂夾定點
      OR      M7085
      OUT     T2630 K10
      MPS
      AND     T2630
      OUT     M7073  ; 回上位Panel#1出板訊號
      MPP
      OUT     T2631 K5
      AND     T2631
      MEP
      SET     M6110  ; 回上位Panel生產結束訊號
; [Title]SECS_時間同步功能
; ********* PLC 系統時間修改 **********
622   LD      SM400  ; Run On
      OUT     SM213
      BMOV    SD210 ZR15000 K4
628   LD      SM400  ; Run On
      WAND    ZR15000 H0FF00 ZR15010
      ROR     ZR15010 K8
        [note] 高低位資料互換
      WAND    ZR15000 H0FF ZR15011
648   LD      SM400  ; Run On
      WAND    ZR15001 H0FF00 ZR15012
      ROR     ZR15012 K8
        [note] 高低位資料互換
      WAND    ZR15001 H0FF ZR15004
      ROR     ZR15004 K8
        [note] 高低位資料互換
681   LD      SM400  ; Run On
      WAND    ZR15002 H0FF00 ZR15005
      ROR     ZR15005 K8
        [note] 高低位資料互換
      WOR     ZR15004 ZR15005 ZR15013
701   LD      M6015  ; SECS_上位下寫入時間
      ANI     ZR15006.0
      SET     ZR15006.0
      MOVP    K0 ZR15007
707   LD<=    ZR15007 K1
      AND     SM412  ; 1.0 Sec Clock
      INCP    ZR15007
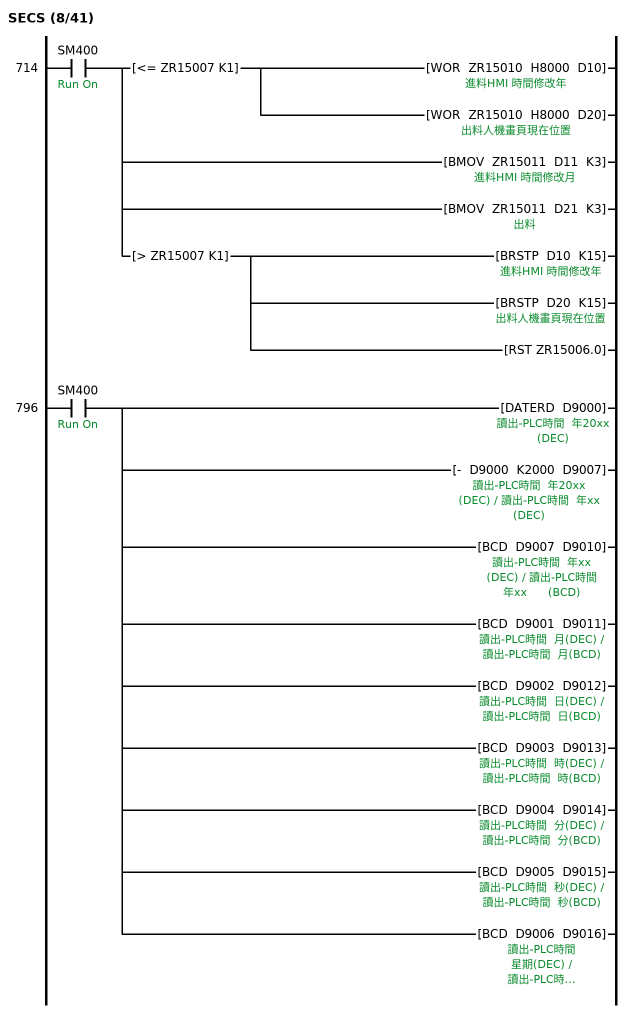
714   LD      SM400  ; Run On
      MPS
      AND<=   ZR15007 K1
      WOR     ZR15010 H8000 D10  ; 進料HMI 時間修改年
        [note] HMI 時間修改命令H8000
      WOR     ZR15010 H8000 D20
        [note] HMI 時間修改命令H8000
      MPP
      BMOV    ZR15011 D11 K3  ; 進料HMI 時間修改月
      BMOV    ZR15011 D21 K3  ; 出料
      AND>    ZR15007 K1
      BRSTP   D10 K15
        [note] HMI 時間修改命令解除
      BRSTP   D20 K15
        [note] HMI 時間修改命令解除
      RST     ZR15006.0
796   LD      SM400  ; Run On
      DATERD  D9000  ; 讀出-PLC時間  年20xx    (DEC)
      -       D9000 K2000 D9007  ; 讀出-PLC時間  年xx      (DEC)
      BCD     D9007 D9010  ; 讀出-PLC時間  年xx      (BCD)
      BCD     D9001 D9011  ; 讀出-PLC時間  月(DEC) / 讀出-PLC時間  月(BCD)
      BCD     D9002 D9012  ; 讀出-PLC時間  日(DEC) / 讀出-PLC時間  日(BCD)
      BCD     D9003 D9013  ; 讀出-PLC時間  時(DEC) / 讀出-PLC時間  時(BCD)
      BCD     D9004 D9014  ; 讀出-PLC時間  分(DEC) / 讀出-PLC時間  分(BCD)
      BCD     D9005 D9015  ; 讀出-PLC時間  秒(DEC) / 讀出-PLC時間  秒(BCD)
      BCD     D9006 D9016  ; 讀出-PLC時間  星期(DEC) / 讀出-PLC時間  星期(BCD)
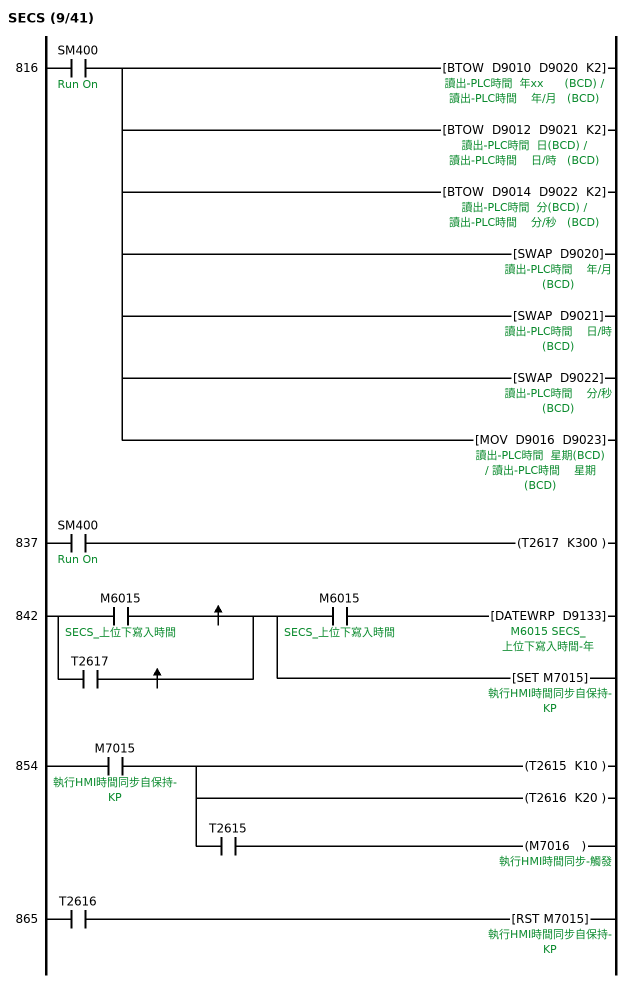
816   LD      SM400  ; Run On
      BTOW    D9010 D9020 K2  ; 讀出-PLC時間    年/月   (BCD)
      BTOW    D9012 D9021 K2  ; 讀出-PLC時間    日/時   (BCD)
      BTOW    D9014 D9022 K2  ; 讀出-PLC時間    分/秒   (BCD)
      SWAP    D9020
      SWAP    D9021
      SWAP    D9022
      MOV     D9016 D9023  ; 讀出-PLC時間    星期    (BCD)
837   LD      SM400  ; Run On
      OUT     T2617 K300
842   LD      M6015  ; SECS_上位下寫入時間
      MEP
      LD      T2617
      MEP
      ORB
      MPS
      AND     M6015  ; SECS_上位下寫入時間
      DATEWRP D9133  ; M6015 SECS_上位下寫入時間-年
      MPP
      SET     M7015  ; 執行HMI時間同步自保持-KP
854   LD      M7015  ; 執行HMI時間同步自保持-KP
      OUT     T2615 K10
      OUT     T2616 K20
      AND     T2615
      OUT     M7016  ; 執行HMI時間同步-觸發
865   LD      T2616
      RST     M7015  ; 執行HMI時間同步自保持-KP
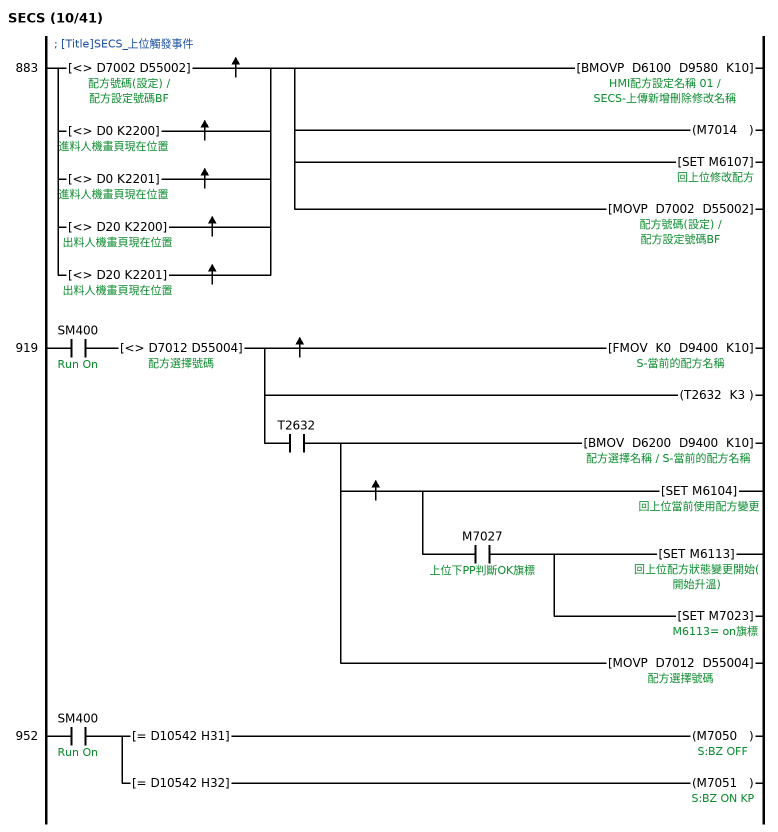
; [Title]SECS_上位觸發事件
883   LD<>    D7002 D55002  ; 配方號碼(設定) / 配方設定號碼BF
      MEP
      LD<>    D0 K2200  ; 進料人機畫頁現在位置
      MEP
      ORB
      LD<>    D0 K2201  ; 進料人機畫頁現在位置
      MEP
      ORB
      LD<>    D20 K2200  ; 出料人機畫頁現在位置
      MEP
      ORB
      LD<>    D20 K2201  ; 出料人機畫頁現在位置
      MEP
      ORB
      BMOVP   D6100 D9580 K10  ; HMI配方設定名稱 01 / SECS-上傳新增刪除修改名稱
      OUT     M7014
      SET     M6107  ; 回上位修改配方
      MOVP    D7002 D55002
919   LD      SM400  ; Run On
      AND<>   D7012 D55004  ; 配方選擇號碼
      MPS
      MEP
      FMOV    K0 D9400 K10  ; S-當前的配方名稱
      MPP
      OUT     T2632 K3
      AND     T2632
      BMOV    D6200 D9400 K10  ; 配方選擇名稱
      MPS
      MEP
      SET     M6104  ; 回上位當前使用配方變更
      AND     M7027  ; 上位下PP判斷OK旗標
      SET     M6113  ; 回上位配方狀態變更開始(開始升溫)
      SET     M7023  ; M6113= on旗標
      MPP
      MOVP    D7012 D55004
952   LD      SM400  ; Run On
      MPS
      AND=    D10542 H31
      OUT     M7050  ; S:BZ OFF
      MPP
      AND=    D10542 H32
      OUT     M7051  ; S:BZ ON KP
